(* IEC 61131-3 sources: B-R/Processes/EDT (part 3) *)

(* ---- EDTP3S2A_ACTION.st ---- *)
ACTION P3S2A_ACT:
	//设定时间
	FOR i := 0 TO EDTP3S2_STEP_NUM DO
		IF EDTP3S2A_ST[i] < T#5s THEN
			EDTP3S2A_ST[i] := T#5s;
		END_IF;
		EDTP3S2A_STEP[i].set_time := EDTP3S2A_ST[i];
	END_FOR;

	//流程步骤
	ProcessHandleFC(EDTP3S2A,EDTP3S2A_STEP[0],EDTP3S2_STEP_NUM);

	//object 手自动切换
	IF (EDTP3S2A.status.mode <> 0) AND (NOT EDTP3S2A.auto_mode_edge) THEN
		EDTP3S2A.auto_mode_edge := TRUE;
		EDTP3S2A.manual_mode_edge := FALSE;

		EDTR17A.control.auto_operate := TRUE;
		EDTXV0902.control.auto_operate := TRUE;
		EDTXV2128.control.auto_operate := TRUE;
		EDTXV2119.control.auto_operate := TRUE;
		EDTXV2121.control.auto_operate := TRUE;
		EDTTV0901C.control.auto_operate := TRUE;
		EDTTV0901D.control.auto_operate := TRUE;
		EDTTV0901E.control.auto_operate := TRUE;
		EDTTV0901F.control.auto_operate := TRUE;
		EDTTV0902B.control.auto_operate := TRUE;
		EDTTV0902A.control.auto_operate := TRUE;
		EDTTV0901A.control.auto_operate := TRUE;
		EDTTV0901B.control.auto_operate := TRUE;
		EDTXV0918.control.auto_operate := TRUE;
		EDTFQV0901.control.auto_operate := TRUE;
		EDTFQV0904.control.auto_operate := TRUE;
		EDTLV1002.control.auto_operate := TRUE;
		EDTP16.control.auto_operate := TRUE;
		EDTXV0925.control.auto_operate := TRUE;
		STFP06.control.auto_operate := TRUE;
		STFLV0601.control.auto_operate := TRUE;
		STFLV0602.control.auto_operate := TRUE;
		EDTLV1003.control.auto_operate := TRUE;
	END_IF;

	IF (EDTP3S2A.status.mode = 0) AND (NOT EDTP3S2A.manual_mode_edge) THEN
		EDTP3S2A.manual_mode_edge := TRUE;
		EDTP3S2A.auto_mode_edge := FALSE;

		EDTR17A.control.manual_operate := TRUE;
		EDTXV0902.control.manual_operate := TRUE;
		EDTXV2128.control.manual_operate := TRUE;
		EDTXV2119.control.manual_operate := TRUE;
		EDTXV2121.control.manual_operate := TRUE;
		EDTTV0901C.control.manual_operate := TRUE;
		EDTTV0901D.control.manual_operate := TRUE;
		EDTTV0901E.control.manual_operate := TRUE;
		EDTTV0901F.control.manual_operate := TRUE;
		EDTTV0902B.control.manual_operate := TRUE;
		EDTTV0902A.control.manual_operate := TRUE;
		EDTTV0901A.control.manual_operate := TRUE;
		EDTTV0901B.control.manual_operate := TRUE;
		EDTXV0918.control.manual_operate := TRUE;
		EDTFQV0901.control.manual_operate := TRUE;
		EDTFQV0904.control.manual_operate := TRUE;
		EDTLV1002.control.manual_operate := TRUE;
		EDTP16.control.manual_operate := TRUE;
		EDTXV0925.control.manual_operate := TRUE;
		STFP06.control.manual_operate := TRUE;
		STFLV0601.control.manual_operate := TRUE;
		STFLV0602.control.manual_operate := TRUE;
		EDTLV1003.control.manual_operate := TRUE;
	END_IF;

	//错误信号停机
	EDTP3S2A.input.error_signal := (EDTR17A.status.motor_status >= 2) OR (EDTXV0902.status.valve_status >= 2) OR
	(EDTXV2128.status.valve_status >= 2) OR (EDTXV2119.status.valve_status >= 2) OR (EDTP16.status.motor_status >= 2) OR
	(EDTTV0901C.status.valve_status >= 2) OR (EDTTV0901D.status.valve_status >= 2) OR (EDTXV0918.status.valve_status >= 2) OR
	(EDTTV0901E.status.valve_status >= 2) OR (EDTTV0901F.status.valve_status >= 2) OR (EDTTV0902B.status.valve_status >= 2) OR
	(EDTTV0902A.status.valve_status >= 2) OR (EDTTV0901A.status.valve_status >= 2) OR (EDTTV0901B.status.valve_status >= 2) OR
	(EDTFQV0901.status.valve_status >= 2) OR (EDTFQV0904.status.valve_status >= 2) OR (EDTLV1002.status.valve_status >= 2) OR
	(EDTXV2121.status.valve_status >= 2) OR (EDTXV0925.status.valve_status >= 2) OR (STFP06.status.motor_status >= 2) OR
	(EDTLV1003.status.valve_status >= 2) OR (STFLV0601.status.valve_status >= 2 )OR (STFLV0602.status.valve_status >= 2);

	IF EDTP3S2A.status.run_state = 1 THEN
		CASE EDTP3S2A.status.run_step OF
			0:
				IF NOT EDTP3S2A_STEP[0].done THEN
					EDTR17A.control.auto_operate := TRUE;
					EDTXV0902.control.auto_operate := TRUE;
					EDTXV2128.control.auto_operate := TRUE;
					EDTXV2119.control.auto_operate := TRUE;
					EDTXV2121.control.auto_operate := TRUE;
					EDTTV0901C.control.auto_operate := TRUE;
					EDTTV0901D.control.auto_operate := TRUE;
					EDTTV0901E.control.auto_operate := TRUE;
					EDTTV0901F.control.auto_operate := TRUE;
					EDTTV0902B.control.auto_operate := TRUE;
					EDTTV0902A.control.auto_operate := TRUE;
					EDTTV0901A.control.auto_operate := TRUE;
					EDTTV0901B.control.auto_operate := TRUE;
					EDTXV0918.control.auto_operate := TRUE;
					EDTFQV0901.control.auto_operate := TRUE;
					EDTFQV0904.control.auto_operate := TRUE;
					EDTLV1002.control.auto_operate := TRUE;
					EDTP16.control.auto_operate := TRUE;
					EDTXV0925.control.auto_operate := TRUE;
					STFP06.control.auto_operate := TRUE;
					STFLV0601.control.auto_operate := TRUE;
					STFLV0602.control.auto_operate := TRUE;
					EDTLV1003.control.auto_operate := TRUE;
					EDTP3S2A_STEP[0].done := TRUE;
				END_IF;
			1:
				EDTXV0925.input.auto_open_signal := TRUE;
				IF EDTXV0905.input.close_feedback_state THEN
					EDTR17A.input.auto_run_signal := TRUE;
					EDTXV0902.input.auto_open_signal := TRUE;
					EDTTV0902A.input.auto_open_signal := FALSE;
					EDTXV2128.input.auto_open_signal := FALSE;
					IF EDTTV0902A.input.close_feedback_state AND EDTXV2128.input.close_feedback_state THEN
						EDTTV0902B.input.auto_open_signal := TRUE;
						IF EDTR17A.input.run_feedback AND EDTXV0902.input.open_feedback_state AND EDTTV0902B.input.open_feedback_state THEN
							EDTP3S2A_STEP[1].done := TRUE;
						END_IF;
					END_IF;
				END_IF;
			2:
				CASE p3_step2_3a OF
					0:
						IF NOT EDTP3S2A_STEP[2].done THEN
							p3_step2_3a := 1;
						END_IF;
					1:
						HeatPot_1(ST1 := DINT_TO_TIME(EDTP3S2A_PARA_T1 * 1000),
						ST2 := DINT_TO_TIME(EDTP3S2A_PARA_T2 * 1000),
						V3 := EDTTV0901C,
						V4 := EDTTV0901D,
						V5 := EDTTV0901E,
						V6 := EDTTV0901F,
						done := p3_step2_3a_1_done);
						IF p3_step2_3a_1_done THEN
							p3_step2_3a_1_done := FALSE;
							p3_step2_3a := 2;
						END_IF;
					2:
						IF EDTTIT0901.status.value >= EDTP3S2A_PARA_Temp1 THEN
							p3_step2_3a := 3;
						END_IF;
					3:
						EDTTV0901C.input.auto_open_signal := FALSE;
						IF EDTTV0901C.input.close_feedback_state THEN
							p3_step2_3a := 4;
						END_IF;
					4:
						IF EDTLIT0901.status.value >= EDTP3S2A_PARA_L1 THEN
							EDTTV0902B.input.auto_open_signal := FALSE;
							EDTTV0902A.input.auto_open_signal := TRUE;
							IF EDTXV2128.input.close_feedback_state THEN
								EDTXV0918.input.auto_open_signal := TRUE;
							END_IF;
							p3_step2_3a := 5;
						END_IF;
					5:
						IF EDTXV2128.input.open_feedback_state THEN
							EDTXV0918.input.auto_open_signal := FALSE;
						END_IF;
						IF EDTTIT0901.status.value >= EDTP3S2A_PARA_Temp2 THEN
							EDTXV0918.input.auto_open_signal := FALSE;
							EDTXV2128.input.auto_open_signal := TRUE;
							EDTXV2119.input.auto_open_signal := TRUE;
							EDTXV2121.input.auto_open_signal := TRUE;
							p3_step2_3a := 0;
							EDTP3S2A_STEP[2].done := TRUE;
						END_IF;
				END_CASE;
			3:
				LiquidTransfer_12(sp_time := DINT_TO_TIME(EDTP3S2A_PARA_T4 * 1000),
				sp_accumulation := EDTP3S2A_PARA_AC1,
				done := EDTP3S2A_STEP[3].done,
				flowmeter := EDTFQIT1904);
				EDTFQV0901.input.auto_open_signal := LiquidTransfer_12.run;
			4:
				//继续回收
				IF EDTTIT0901.status.value >= EDTP3S2A_PARA_Temp3 THEN
					EDTP3S2A_STEP[4].done := TRUE;
				END_IF;
			5:
				//现场观察V83进料的是否有EDC油珠，无油珠后点击确认
			6:
				EDTTV0901D.input.auto_open_signal := FALSE;
				EDTTV0901E.input.auto_open_signal := FALSE;
				EDTTV0901F.input.auto_open_signal := TRUE;
				LiquidTransfer_16(sp_time := DINT_TO_TIME(EDTP3S2A_PARA_T5 * 1000),
				sp_accumulation := EDTP3S2A_PARA_AC2,
				done := EDTP3S2A_STEP[6].done,
				flowmeter := EDTFQIT1904);
				EDTFQV0901.input.auto_open_signal := LiquidTransfer_16.run;
			7:
				CASE p3_step2_7a OF
					0:
						IF NOT EDTP3S2A_STEP[7].done THEN
							p3_step2_7a := 1;
						END_IF;
					1:
						IF EDTTIT0901.status.value <= EDTP3S2A_PARA_Temp6 THEN
							EDTTV0901A.input.auto_open_signal := FALSE;
							EDTTV0901B.input.auto_open_signal := FALSE;
							EDTTV0901F.input.auto_open_signal := TRUE;
							p3_step2_7a := 2;
						ELSE
							EDTTV0901F.input.auto_open_signal := FALSE;
							EDTTV0901A.input.auto_open_signal := TRUE;
							EDTTV0901B.input.auto_open_signal := TRUE;
						END_IF;
					2:
						TON_60.PT := DINT_TO_TIME(EDTP3S2A_PARA_T9 * 60 * 1000);
						EDTR17A.input.auto_run_signal := FALSE;
						IF (NOT EDTR17A.input.run_feedback) THEN
							TON_60.IN := TRUE;
						END_IF;
						IF TON_60.Q THEN
							TON_60.IN := FALSE;
							p3_step2_7a := 0;
							EDTP3S2A_STEP[7].done := TRUE;
						END_IF;
				END_CASE;
				TON_60();
			8:
				//人工抽水,完毕后点击确认
			9:
				IF EDTLIT1501.status.value >= EDTP3S2A_PARA_L2 THEN
					EDTFQV0904.input.auto_open_signal := TRUE;
					EDTLV1002.input.auto_open_signal := TRUE;
					IF EDTFQV0904.input.open_feedback_state AND EDTLV1002.input.open_feedback_state THEN
						is_v52_a := TRUE;
						EDTP3S2A_STEP[9].done := TRUE;
					END_IF;
				ELSE
					STFLV0601.input.auto_open_signal := FALSE;
					STFLV0602.input.auto_open_signal := FALSE;
					EDTFQV0904.input.auto_open_signal := TRUE;
					EDTLV1003.input.auto_open_signal := TRUE;
					IF STFLV0601.input.close_feedback_state AND STFLV0602.input.close_feedback_state AND EDTFQV0904.input.open_feedback_state AND EDTLV1003.input.open_feedback_state THEN
						is_v52_a := FALSE;
						EDTP3S2A_STEP[9].done := TRUE;
					END_IF;
				END_IF;
			10:
				IF is_v52_a THEN
					LiquidTransfer_21(sp_time := DINT_TO_TIME(EDTP3S2A_PARA_T6 * 1000),
					sp_accumulation := EDTP3S2A_PARA_AC3,
					done := EDTP3S2A_STEP[10].done,
					flowmeter := EDTFQIT2101);
					EDTP16.input.auto_run_signal := LiquidTransfer_21.run;
				ELSE
					LiquidTransfer_1(sp_time := DINT_TO_TIME(EDTP3S2A_PARA_T6 * 1000),
					sp_accumulation := EDTP3S2A_PARA_AC3,
					done := EDTP3S2A_STEP[10].done,
					flowmeter := STFFQIT0602);
					STFP06.input.auto_run_signal := LiquidTransfer_1.run;
				END_IF;
			11:
				IF is_v52_a THEN
					IF EDTFQIT2101.flowrate <= flowrate_threshold THEN
						EDTFQV0904.input.auto_open_signal := FALSE;
						EDTLV1002.input.auto_open_signal := FALSE;
						EDTR17A.input.auto_run_signal := TRUE;
						IF EDTFQV0904.input.close_feedback_state AND EDTLV1002.input.close_feedback_state AND EDTR17A.input.auto_run_signal THEN
							EDTTV0901D.input.auto_open_signal := TRUE;
							EDTP3S2A_STEP[11].done := TRUE;
						END_IF;
					END_IF;
				ELSE
					IF STFFQIT0602.flowrate <= flowrate_threshold THEN
						EDTFQV0904.input.auto_open_signal := FALSE;
						EDTLV1003.input.auto_open_signal := FALSE;
						EDTR17A.input.auto_run_signal := TRUE;
						IF EDTFQV0904.input.close_feedback_state AND EDTLV1003.input.close_feedback_state AND EDTR17A.input.auto_run_signal THEN
							EDTTV0901D.input.auto_open_signal := TRUE;
							EDTP3S2A_STEP[11].done := TRUE;
						END_IF;
					END_IF;
				END_IF;

			12:
				TON_21.PT := DINT_TO_TIME(EDTP3S2A_PARA_T7 * 1000);
				IF EDTTV0901D.input.open_feedback_state THEN
					TON_21.IN := TRUE;
				END_IF;
				IF TON_21.Q THEN
					TON_21.IN := FALSE;
					EDTTV0901F.input.auto_open_signal := FALSE;
					EDTTV0901E.input.auto_open_signal := TRUE;
					EDTP3S2A_STEP[12].done := TRUE;
				END_IF;
				TON_21();
			13:
				TON_26.PT := DINT_TO_TIME(EDTP3S2A_PARA_T8 * 60 * 1000);
				IF EDTTIT0901.status.value >= EDTP3S2A_PARA_Temp4 THEN
					EDTTV0901D.input.auto_open_signal := FALSE;
					TON_26.IN := TRUE;
				END_IF;
				IF TON_26.Q THEN
					TON_26.IN := FALSE;
					EDTP3S2A_STEP[13].done := TRUE;
				END_IF;
				TON_26();
			14:
				//人工转移
			15:
				EDTR17A.input.auto_run_signal := FALSE;
				EDTTV0901E.input.auto_open_signal := FALSE;
				EDTP3S2A_STEP[15].done := TRUE;
		END_CASE;
	END_IF;

	//人工确认步骤可用
	IF (EDTP3S2A.status.run_state) AND (NOT EDTP3S2A_STEP[EDTP3S2A.status.run_step].done AND ((EDTP3S2A.status.run_step = 5)
		OR (EDTP3S2A.status.run_step = 8) OR (EDTP3S2A.status.run_step = 14))) THEN
		EDTP3S2A.status.confirm_enable := TRUE;
	ELSE
		EDTP3S2A.status.confirm_enable := FALSE;
	END_IF;
END_ACTION

(* ---- EDTP3S2B_ACTION.st ---- *)
ACTION P3S2B_ACT:
	//设定时间
	FOR i := 0 TO EDTP3S2_STEP_NUM DO
		IF EDTP3S2B_ST[i] < T#5s THEN
			EDTP3S2B_ST[i] := T#5s;
		END_IF;
		EDTP3S2B_STEP[i].set_time := EDTP3S2B_ST[i];
	END_FOR;

	//流程步骤
	ProcessHandleFC(EDTP3S2B,EDTP3S2B_STEP[0],EDTP3S2_STEP_NUM);

	//object 手自动切换
	IF (EDTP3S2B.status.mode <> 0) AND (NOT EDTP3S2B.auto_mode_edge) THEN
		EDTP3S2B.auto_mode_edge := TRUE;
		EDTP3S2B.manual_mode_edge := FALSE;

		EDTR17B.control.auto_operate := TRUE;
		EDTXV0912.control.auto_operate := TRUE;
		EDTXV2128.control.auto_operate := TRUE;
		EDTXV2119.control.auto_operate := TRUE;
		EDTXV2121.control.auto_operate := TRUE;
		EDTTV0903C.control.auto_operate := TRUE;
		EDTTV0903D.control.auto_operate := TRUE;
		EDTTV0903E.control.auto_operate := TRUE;
		EDTTV0903F.control.auto_operate := TRUE;
		EDTTV0904B.control.auto_operate := TRUE;
		EDTTV0904A.control.auto_operate := TRUE;
		EDTTV0903A.control.auto_operate := TRUE;
		EDTTV0903B.control.auto_operate := TRUE;
		EDTXV0918.control.auto_operate := TRUE;
		EDTFQV0902.control.auto_operate := TRUE;
		EDTFQV0905.control.auto_operate := TRUE;
		EDTLV1002.control.auto_operate := TRUE;
		EDTP16.control.auto_operate := TRUE;
		EDTXV0925.control.auto_operate := TRUE;
		STFP06.control.auto_operate := TRUE;
		STFLV0601.control.auto_operate := TRUE;
		STFLV0602.control.auto_operate := TRUE;
		EDTLV1003.control.auto_operate := TRUE;
	END_IF;

	IF (EDTP3S2B.status.mode = 0) AND (NOT EDTP3S2B.manual_mode_edge) THEN
		EDTP3S2B.manual_mode_edge := TRUE;
		EDTP3S2B.auto_mode_edge := FALSE;

		EDTR17B.control.manual_operate := TRUE;
		EDTXV0912.control.manual_operate := TRUE;
		EDTXV2128.control.manual_operate := TRUE;
		EDTXV2119.control.manual_operate := TRUE;
		EDTXV2121.control.manual_operate := TRUE;
		EDTTV0903C.control.manual_operate := TRUE;
		EDTTV0903D.control.manual_operate := TRUE;
		EDTTV0903E.control.manual_operate := TRUE;
		EDTTV0903F.control.manual_operate := TRUE;
		EDTTV0904B.control.manual_operate := TRUE;
		EDTTV0904A.control.manual_operate := TRUE;
		EDTTV0903A.control.manual_operate := TRUE;
		EDTTV0903B.control.manual_operate := TRUE;
		EDTXV0918.control.manual_operate := TRUE;
		EDTFQV0902.control.manual_operate := TRUE;
		EDTFQV0905.control.manual_operate := TRUE;
		EDTLV1002.control.manual_operate := TRUE;
		EDTP16.control.manual_operate := TRUE;
		EDTXV0925.control.manual_operate := TRUE;
		STFP06.control.manual_operate := TRUE;
		STFLV0601.control.manual_operate := TRUE;
		STFLV0602.control.manual_operate := TRUE;
		EDTLV1003.control.manual_operate := TRUE;
	END_IF;

	//错误信号停机
	EDTP3S2B.input.error_signal := (EDTR17B.status.motor_status >= 2) OR (EDTXV0912.status.valve_status >= 2) OR
	(EDTXV2128.status.valve_status >= 2) OR (EDTXV2119.status.valve_status >= 2) OR (EDTP16.status.motor_status >= 2) OR
	(EDTTV0903C.status.valve_status >= 2) OR (EDTTV0903D.status.valve_status >= 2) OR (EDTXV0918.status.valve_status >= 2) OR
	(EDTTV0903E.status.valve_status >= 2) OR (EDTTV0903F.status.valve_status >= 2) OR (EDTTV0904B.status.valve_status >= 2) OR
	(EDTTV0904A.status.valve_status >= 2) OR (EDTTV0903A.status.valve_status >= 2) OR (EDTTV0903B.status.valve_status >= 2) OR
	(EDTFQV0902.status.valve_status >= 2) OR (EDTFQV0905.status.valve_status >= 2) OR (EDTLV1002.status.valve_status >= 2) OR
	(EDTXV2121.status.valve_status >= 2) OR (EDTXV0925.status.valve_status >= 2) OR (STFP06.status.motor_status >= 2) OR
	(EDTLV1003.status.valve_status >= 2) OR (STFLV0601.status.valve_status >= 2 )OR (STFLV0602.status.valve_status >= 2);

	IF EDTP3S2B.status.run_state = 1 THEN
		CASE EDTP3S2B.status.run_step OF
			0:
				IF NOT EDTP3S2B_STEP[0].done THEN
					EDTR17B.control.auto_operate := TRUE;
					EDTXV0912.control.auto_operate := TRUE;
					EDTXV2128.control.auto_operate := TRUE;
					EDTXV2119.control.auto_operate := TRUE;
					EDTXV2121.control.auto_operate := TRUE;
					EDTTV0903C.control.auto_operate := TRUE;
					EDTTV0903D.control.auto_operate := TRUE;
					EDTTV0903E.control.auto_operate := TRUE;
					EDTTV0903F.control.auto_operate := TRUE;
					EDTTV0904B.control.auto_operate := TRUE;
					EDTTV0904A.control.auto_operate := TRUE;
					EDTTV0903A.control.auto_operate := TRUE;
					EDTTV0903B.control.auto_operate := TRUE;
					EDTXV0918.control.auto_operate := TRUE;
					EDTFQV0902.control.auto_operate := TRUE;
					EDTFQV0905.control.auto_operate := TRUE;
					EDTLV1002.control.auto_operate := TRUE;
					EDTP16.control.auto_operate := TRUE;
					EDTXV0925.control.auto_operate := TRUE;
					STFP06.control.auto_operate := TRUE;
					STFLV0601.control.auto_operate := TRUE;
					STFLV0602.control.auto_operate := TRUE;
					EDTLV1003.control.auto_operate := TRUE;
					EDTP3S2B_STEP[0].done := TRUE;
				END_IF;
			1:
				EDTXV0925.input.auto_open_signal := TRUE;
				IF EDTXV0913.input.close_feedback_state THEN
					EDTR17B.input.auto_run_signal := TRUE;
					EDTXV0912.input.auto_open_signal := TRUE;
					EDTTV0904A.input.auto_open_signal := FALSE;
					EDTXV2128.input.auto_open_signal := FALSE;
					IF EDTTV0904A.input.close_feedback_state AND EDTXV2128.input.close_feedback_state THEN
						EDTTV0904B.input.auto_open_signal := TRUE;
						IF EDTR17B.input.run_feedback AND EDTXV0912.input.open_feedback_state AND EDTTV0904B.input.open_feedback_state THEN
							EDTP3S2B_STEP[1].done := TRUE;
						END_IF;
					END_IF;
				END_IF;
			2:
				CASE p3_step2_3b OF
					0:
						IF NOT EDTP3S2B_STEP[2].done THEN
							p3_step2_3b := 1;
						END_IF;
					1:
						HeatPot_11(ST1 := DINT_TO_TIME(EDTP3S2B_PARA_T1 * 1000),
						ST2 := DINT_TO_TIME(EDTP3S2B_PARA_T2 * 1000),
						V3 := EDTTV0903C,
						V4 := EDTTV0903D,
						V5 := EDTTV0903E,
						V6 := EDTTV0903F,
						done := p3_step2_3b_1_done);
						IF p3_step2_3b_1_done THEN
							p3_step2_3b_1_done := FALSE;
							p3_step2_3b := 2;
						END_IF;
					2:
						IF EDTTIT0903.status.value >= EDTP3S2B_PARA_Temp1 THEN
							p3_step2_3b := 3;
						END_IF;
					3:
						EDTTV0903C.input.auto_open_signal := FALSE;
						IF EDTTV0903C.input.close_feedback_state THEN
							p3_step2_3b := 4;
						END_IF;
					4:
						IF EDTLIT0902.status.value >= EDTP3S2B_PARA_L1 THEN
							EDTTV0904B.input.auto_open_signal := FALSE;
							EDTTV0904A.input.auto_open_signal := TRUE;
							IF EDTXV2128.input.close_feedback_state THEN
								EDTXV0918.input.auto_open_signal := TRUE;
							END_IF;
							p3_step2_3b := 5;
						END_IF;
					5:
						IF EDTXV2128.input.open_feedback_state THEN
							EDTXV0918.input.auto_open_signal := FALSE;
						END_IF;
						IF EDTTIT0903.status.value >= EDTP3S2B_PARA_Temp2 THEN
							EDTXV0918.input.auto_open_signal := FALSE;
							EDTXV2128.input.auto_open_signal := TRUE;
							EDTXV2119.input.auto_open_signal := TRUE;
							EDTXV2121.input.auto_open_signal := TRUE;
							p3_step2_3b := 0;
							EDTP3S2B_STEP[2].done := TRUE;
						END_IF;
				END_CASE;
			3:
				LiquidTransfer_17(sp_time := DINT_TO_TIME(EDTP3S2B_PARA_T4 * 1000),
				sp_accumulation := EDTP3S2B_PARA_AC1,
				done := EDTP3S2B_STEP[3].done,
				flowmeter := EDTFQIT1904);
				EDTFQV0902.input.auto_open_signal := LiquidTransfer_17.run;
			4:
				//继续回收
				IF EDTTIT0903.status.value >= EDTP3S2B_PARA_Temp3 THEN
					EDTP3S2B_STEP[4].done := TRUE;
				END_IF;
			5:
				//现场观察V83进料的是否有EDC油珠，无油珠后点击确认
			6:
				EDTTV0903D.input.auto_open_signal := FALSE;
				EDTTV0903E.input.auto_open_signal := FALSE;
				EDTTV0903F.input.auto_open_signal := TRUE;
				LiquidTransfer_18(sp_time := DINT_TO_TIME(EDTP3S2B_PARA_T5 * 1000),
				sp_accumulation := EDTP3S2B_PARA_AC2,
				done := EDTP3S2B_STEP[6].done,
				flowmeter := EDTFQIT1904);
				EDTFQV0902.input.auto_open_signal := LiquidTransfer_18.run;
			7:
				CASE p3_step2_7b OF
					0:
						IF NOT EDTP3S2B_STEP[7].done THEN
							p3_step2_7b := 1;
						END_IF;
					1:
						IF EDTTIT0903.status.value <= EDTP3S2B_PARA_Temp6 THEN
							EDTTV0903A.input.auto_open_signal := FALSE;
							EDTTV0903B.input.auto_open_signal := FALSE;
							EDTTV0903F.input.auto_open_signal := TRUE;
							p3_step2_7b := 2;
						ELSE
							EDTTV0903F.input.auto_open_signal := FALSE;
							EDTTV0903A.input.auto_open_signal := TRUE;
							EDTTV0903B.input.auto_open_signal := TRUE;
						END_IF;
					2:
						TON_85.PT := DINT_TO_TIME(EDTP3S2B_PARA_T9 * 60 * 1000);
						EDTR17B.input.auto_run_signal := FALSE;
						IF (NOT EDTR17B.input.run_feedback) THEN
							TON_85.IN := TRUE;
						END_IF;
						IF TON_85.Q THEN
							TON_85.IN := FALSE;
							p3_step2_7b := 0;
							EDTP3S2B_STEP[7].done := TRUE;
						END_IF;
				END_CASE;
				TON_85();
			8:
				//人工抽水
			9:
				IF EDTLIT1501.status.value >= EDTP3S2B_PARA_L2 THEN
					EDTFQV0905.input.auto_open_signal := TRUE;
					EDTLV1002.input.auto_open_signal := TRUE;
					IF EDTFQV0905.input.open_feedback_state AND EDTLV1002.input.open_feedback_state THEN
						is_v52_b := TRUE;
						EDTP3S2B_STEP[9].done := TRUE;
					END_IF;
				ELSE
					STFLV0601.input.auto_open_signal := FALSE;
					STFLV0602.input.auto_open_signal := FALSE;
					EDTFQV0905.input.auto_open_signal := TRUE;
					EDTLV1003.input.auto_open_signal := TRUE;
					IF STFLV0601.input.close_feedback_state AND STFLV0602.input.close_feedback_state AND EDTFQV0905.input.open_feedback_state AND EDTLV1003.input.open_feedback_state THEN
						is_v52_b := FALSE;
						EDTP3S2B_STEP[9].done := TRUE;
					END_IF;
				END_IF;
			10:
				IF is_v52_b THEN
					LiquidTransfer_22(sp_time := DINT_TO_TIME(EDTP3S2B_PARA_T6 * 1000),
					sp_accumulation := EDTP3S2B_PARA_AC3,
					done := EDTP3S2B_STEP[10].done,
					flowmeter := EDTFQIT2101);
					EDTP16.input.auto_run_signal := LiquidTransfer_22.run;
				ELSE
					LiquidTransfer_2(sp_time := DINT_TO_TIME(EDTP3S2B_PARA_T6 * 1000),
					sp_accumulation := EDTP3S2B_PARA_AC3,
					done := EDTP3S2B_STEP[10].done,
					flowmeter := STFFQIT0602);
					STFP06.input.auto_run_signal := LiquidTransfer_2.run;
				END_IF;
			11:
				IF is_v52_b THEN
					IF EDTFQIT2101.flowrate <= flowrate_threshold THEN
						EDTFQV0905.input.auto_open_signal := FALSE;
						EDTLV1002.input.auto_open_signal := FALSE;
						EDTR17B.input.auto_run_signal := TRUE;
						IF EDTFQV0905.input.close_feedback_state AND EDTLV1002.input.close_feedback_state AND EDTR17B.input.auto_run_signal THEN
							EDTTV0903D.input.auto_open_signal := TRUE;
							EDTP3S2B_STEP[11].done := TRUE;
						END_IF;
					END_IF;
				ELSE
					IF STFFQIT0602.flowrate <= flowrate_threshold THEN
						EDTFQV0905.input.auto_open_signal := FALSE;
						EDTLV1003.input.auto_open_signal := FALSE;
						EDTR17B.input.auto_run_signal := TRUE;
						IF EDTFQV0905.input.close_feedback_state AND EDTLV1003.input.close_feedback_state AND EDTR17B.input.auto_run_signal THEN
							EDTTV0903D.input.auto_open_signal := TRUE;
							EDTP3S2B_STEP[11].done := TRUE;
						END_IF;
					END_IF;
				END_IF;
			12:
				TON_29.PT := DINT_TO_TIME(EDTP3S2B_PARA_T7 * 1000);
				IF EDTTV0903D.input.open_feedback_state THEN
					TON_29.IN := TRUE;
				END_IF;
				IF TON_29.Q THEN
					TON_29.IN := FALSE;
					EDTTV0903F.input.auto_open_signal := FALSE;
					EDTTV0903E.input.auto_open_signal := TRUE;
					EDTP3S2B_STEP[12].done := TRUE;
				END_IF;
				TON_29();
			13:
				TON_42.PT := DINT_TO_TIME(EDTP3S2B_PARA_T8 * 60 * 1000);
				IF EDTTIT0903.status.value >= EDTP3S2B_PARA_Temp4 THEN
					EDTTV0903D.input.auto_open_signal := FALSE;
					TON_42.IN := TRUE;
				END_IF;
				IF TON_42.Q THEN
					TON_42.IN := FALSE;
					EDTP3S2B_STEP[13].done := TRUE;
				END_IF;
				TON_42();
			14:
				//人工转移
			15:
				EDTR17B.input.auto_run_signal := FALSE;
				EDTTV0903E.input.auto_open_signal := FALSE;
				EDTP3S2B_STEP[15].done := TRUE;
		END_CASE;
	END_IF;

	//人工确认步骤可用
	IF (EDTP3S2B.status.run_state) AND (NOT EDTP3S2B_STEP[EDTP3S2B.status.run_step].done AND ((EDTP3S2B.status.run_step = 5)
		OR (EDTP3S2B.status.run_step = 8) OR (EDTP3S2B.status.run_step = 14))) THEN
		EDTP3S2B.status.confirm_enable := TRUE;
	ELSE
		EDTP3S2B.status.confirm_enable := FALSE;
	END_IF;
END_ACTION

(* ---- EDTP3S2C_ACTION.st ---- *)
ACTION P3S2C_ACT:
	//设定时间
	FOR i := 0 TO EDTP3S2_STEP_NUM DO
		IF EDTP3S2C_ST[i] < T#5s THEN
			EDTP3S2C_ST[i] := T#5s;
		END_IF;
		EDTP3S2C_STEP[i].set_time := EDTP3S2C_ST[i];
	END_FOR;

	//流程步骤
	ProcessHandleFC(EDTP3S2C,EDTP3S2C_STEP[0],EDTP3S2_STEP_NUM);

	//object 手自动切换
	IF (EDTP3S2C.status.mode <> 0) AND (NOT EDTP3S2C.auto_mode_edge) THEN
		EDTP3S2C.auto_mode_edge := TRUE;
		EDTP3S2C.manual_mode_edge := FALSE;

		EDTR20.control.auto_operate := TRUE;
		EDTXV2107.control.auto_operate := TRUE;
		EDTXV2119.control.auto_operate := TRUE;
		EDTXV2110.control.auto_operate := TRUE;
		EDTTV2101C.control.auto_operate := TRUE;
		EDTTV2101D.control.auto_operate := TRUE;
		EDTTV2101E.control.auto_operate := TRUE;
		EDTTV2101F.control.auto_operate := TRUE;
		EDTXV2111.control.auto_operate := TRUE;
		EDTXV2113.control.auto_operate := TRUE;
		EDTTV2101B.control.auto_operate := TRUE;
		EDTTV2101A.control.auto_operate := TRUE;
		EDTXV2112.control.auto_operate := TRUE;
		EDTFQV2102.control.auto_operate := TRUE;
		EDTFQV2101.control.auto_operate := TRUE;
		EDTLV1002.control.auto_operate := TRUE;
		EDTP16.control.auto_operate := TRUE;
		EDTXV2109.control.auto_operate := TRUE;
		STFP06.control.auto_operate := TRUE;
		STFLV0601.control.auto_operate := TRUE;
		STFLV0602.control.auto_operate := TRUE;
		EDTLV1003.control.auto_operate := TRUE;
	END_IF;

	IF (EDTP3S2C.status.mode = 0) AND (NOT EDTP3S2C.manual_mode_edge) THEN
		EDTP3S2C.manual_mode_edge := TRUE;
		EDTP3S2C.auto_mode_edge := FALSE;

		EDTR20.control.manual_operate := TRUE;
		EDTXV2107.control.manual_operate := TRUE;
		EDTXV2119.control.manual_operate := TRUE;
		EDTXV2110.control.manual_operate := TRUE;
		EDTTV2101C.control.manual_operate := TRUE;
		EDTTV2101D.control.manual_operate := TRUE;
		EDTTV2101E.control.manual_operate := TRUE;
		EDTTV2101F.control.manual_operate := TRUE;
		EDTXV2111.control.manual_operate := TRUE;
		EDTXV2113.control.manual_operate := TRUE;
		EDTTV2101B.control.manual_operate := TRUE;
		EDTTV2101A.control.manual_operate := TRUE;
		EDTXV2112.control.manual_operate := TRUE;
		EDTFQV2102.control.manual_operate := TRUE;
		EDTFQV2101.control.manual_operate := TRUE;
		EDTLV1002.control.manual_operate := TRUE;
		EDTXV2109.control.manual_operate := TRUE;
		EDTP16.control.manual_operate := TRUE;
		STFP06.control.manual_operate := TRUE;
		STFLV0601.control.manual_operate := TRUE;
		STFLV0602.control.manual_operate := TRUE;
		EDTLV1003.control.manual_operate := TRUE;
	END_IF;

	//错误信号停机
	EDTP3S2C.input.error_signal := (EDTR20.status.motor_status >= 2) OR (EDTXV2107.status.valve_status >= 2) OR
	(EDTXV2119.status.valve_status >= 2) OR (EDTXV2110.status.valve_status >= 2) OR (EDTP16.status.motor_status >= 2) OR
	(EDTTV2101C.status.valve_status >= 2) OR (EDTTV2101D.status.valve_status >= 2) OR (EDTXV2113.status.valve_status >= 2) OR
	(EDTTV2101E.status.valve_status >= 2) OR (EDTTV2101F.status.valve_status >= 2) OR (EDTXV2111.status.valve_status >= 2) OR
	(EDTTV2101B.status.valve_status >= 2) OR (EDTTV2101A.status.valve_status >= 2) OR (STFP06.status.motor_status >= 2) OR
	(EDTFQV2102.status.valve_status >= 2) OR (EDTFQV2101.status.valve_status >= 2) OR (EDTLV1002.status.valve_status >= 2) OR
	(EDTXV2112.status.valve_status >= 2) OR (EDTXV2109.status.valve_status >= 2 )OR (EDTLV1003.status.valve_status >= 2) OR
	(STFLV0601.status.valve_status >= 2 )OR (STFLV0602.status.valve_status >= 2);

	TON_19.PT := DINT_TO_TIME(EDTP3S2C_PARA_T3 * 60 * 1000);
	IF EDTP3S2C.status.run_state = 1 THEN
		IF EDTTIT2102.status.value >= EDTP3S2C_PARA_Temp5 THEN
			TON_19.IN := TRUE;
		END_IF;
		CASE EDTP3S2C.status.run_step OF
			0:
				IF NOT EDTP3S2C_STEP[0].done THEN
					EDTR20.control.auto_operate := TRUE;
					EDTXV2107.control.auto_operate := TRUE;
					EDTXV2119.control.auto_operate := TRUE;
					EDTXV2110.control.auto_operate := TRUE;
					EDTTV2101C.control.auto_operate := TRUE;
					EDTTV2101D.control.auto_operate := TRUE;
					EDTTV2101E.control.auto_operate := TRUE;
					EDTTV2101F.control.auto_operate := TRUE;
					EDTXV2111.control.auto_operate := TRUE;
					EDTXV2113.control.auto_operate := TRUE;
					EDTTV2101B.control.auto_operate := TRUE;
					EDTTV2101A.control.auto_operate := TRUE;
					EDTXV2112.control.auto_operate := TRUE;
					EDTFQV2102.control.auto_operate := TRUE;
					EDTFQV2101.control.auto_operate := TRUE;
					EDTLV1002.control.auto_operate := TRUE;
					EDTP16.control.auto_operate := TRUE;
					EDTXV2109.control.auto_operate := TRUE;
					STFP06.control.auto_operate := TRUE;
					STFLV0601.control.auto_operate := TRUE;
					STFLV0602.control.auto_operate := TRUE;
					EDTLV1003.control.auto_operate := TRUE;
					EDTP3S2C_STEP[0].done := TRUE;
				END_IF;
			1:
				EDTXV2109.input.auto_open_signal := TRUE;
				IF EDTXV2114.input.close_feedback_state THEN
					EDTR20.input.auto_run_signal := TRUE;
					EDTXV2107.input.auto_open_signal := TRUE;
					EDTXV2113.input.auto_open_signal := FALSE;
					IF EDTXV2113.input.close_feedback_state THEN
						EDTXV2111.input.auto_open_signal := TRUE;
						IF EDTR20.input.run_feedback AND EDTXV2107.input.open_feedback_state AND EDTXV2111.input.open_feedback_state THEN
							EDTP3S2C_STEP[1].done := TRUE;
						END_IF;
					END_IF;
				END_IF;
			2:
				CASE p3_step2_3c OF
					0:
						IF NOT EDTP3S2C_STEP[2].done THEN
							p3_step2_3c := 1;
						END_IF;
					1:
						HeatPot_15(ST1 := DINT_TO_TIME(EDTP3S2C_PARA_T1 * 1000),
						ST2 := DINT_TO_TIME(EDTP3S2C_PARA_T2 * 1000),
						V3 := EDTTV2101C,
						V4 := EDTTV2101D,
						V5 := EDTTV2101E,
						V6 := EDTTV2101F,
						done := p3_step2_3c_1_done);
						IF p3_step2_3c_1_done THEN
							p3_step2_3c_1_done := FALSE;
							p3_step2_3c := 2;
						END_IF;
					2:
						IF EDTTIT2101.status.value >= EDTP3S2C_PARA_Temp1 THEN
							p3_step2_3c := 3;
						END_IF;
					3:
						EDTTV2101C.input.auto_open_signal := FALSE;
						IF EDTTV2101C.input.close_feedback_state THEN
							p3_step2_3c := 4;
						END_IF;
					4:
						IF TON_19.Q OR EDTLSS2101.low THEN
							TON_19.IN := FALSE;
							EDTXV2111.input.auto_open_signal := FALSE;
							EDTXV2112.input.auto_open_signal := TRUE;
							p3_step2_3c := 5;
						END_IF
					5:
						IF EDTTIT2101.status.value >= EDTP3S2C_PARA_Temp2 THEN
							EDTXV2112.input.auto_open_signal := FALSE;
							EDTXV2113.input.auto_open_signal := TRUE;
							EDTXV2119.input.auto_open_signal := TRUE;
							EDTXV2110.input.auto_open_signal := TRUE;
							p3_step2_3c := 0;
							EDTP3S2C_STEP[2].done := TRUE;
						END_IF;
				END_CASE;
			3:
				LiquidTransfer_19(sp_time := DINT_TO_TIME(EDTP3S2C_PARA_T4 * 1000),
				sp_accumulation := EDTP3S2C_PARA_AC1,
				done := EDTP3S2C_STEP[3].done,
				flowmeter := EDTFQIT1904);
				EDTFQV2102.input.auto_open_signal := LiquidTransfer_19.run;
			4:
				//继续回收
				IF EDTTIT2101.status.value >= EDTP3S2C_PARA_Temp3 THEN
					EDTP3S2C_STEP[4].done := TRUE;
				END_IF;
			5:
				//现场观察V83进料的是否有EDC油珠，无油珠后点击确认
			6:
				EDTTV2101D.input.auto_open_signal := FALSE;
				EDTTV2101E.input.auto_open_signal := FALSE;
				EDTTV2101F.input.auto_open_signal := TRUE;
				LiquidTransfer_20(sp_time := DINT_TO_TIME(EDTP3S2C_PARA_T5 * 1000),
				sp_accumulation := EDTP3S2C_PARA_AC2,
				done := EDTP3S2C_STEP[6].done,
				flowmeter := EDTFQIT1904);
				EDTFQV2102.input.auto_open_signal := LiquidTransfer_20.run;
			7:
				CASE p3_step2_7c OF
					0:
						IF NOT EDTP3S2C_STEP[7].done THEN
							p3_step2_7c := 1;
						END_IF;
					1:
						IF EDTTIT2101.status.value <= EDTP3S2C_PARA_Temp6 THEN
							EDTTV2101A.input.auto_open_signal := FALSE;
							EDTTV2101B.input.auto_open_signal := FALSE;
							EDTTV2101F.input.auto_open_signal := TRUE;
							p3_step2_7c := 2;
						ELSE
							EDTTV2101F.input.auto_open_signal := FALSE;
							EDTTV2101A.input.auto_open_signal := TRUE;
							EDTTV2101B.input.auto_open_signal := TRUE;
						END_IF;
					2:
						TON_86.PT := DINT_TO_TIME(EDTP3S2C_PARA_T9 * 60 * 1000);
						EDTR20.input.auto_run_signal := FALSE;
						IF (NOT EDTR20.input.run_feedback) THEN
							TON_86.IN := TRUE;
						END_IF;
						IF TON_86.Q THEN
							TON_86.IN := FALSE;
							p3_step2_7c := 0;
							EDTP3S2C_STEP[7].done := TRUE;
						END_IF;
				END_CASE;
				TON_86();
			8:
			//人工抽水
			9:
				IF EDTLIT1501.status.value >= EDTP3S2C_PARA_L2 THEN
					EDTFQV2101.input.auto_open_signal := TRUE;
					EDTLV1002.input.auto_open_signal := TRUE;
					IF EDTFQV2101.input.open_feedback_state AND EDTLV1002.input.open_feedback_state THEN
						is_v52_c := TRUE;
						EDTP3S2C_STEP[9].done := TRUE;
					END_IF;
				ELSE
					STFLV0601.input.auto_open_signal := FALSE;
					STFLV0602.input.auto_open_signal := FALSE;
					EDTFQV2101.input.auto_open_signal := TRUE;
					EDTLV1003.input.auto_open_signal := TRUE;
					IF STFLV0601.input.close_feedback_state AND STFLV0602.input.close_feedback_state AND EDTFQV2101.input.open_feedback_state AND EDTLV1003.input.open_feedback_state THEN
						is_v52_c := FALSE;
						EDTP3S2C_STEP[9].done := TRUE;
					END_IF;
				END_IF;
			10:
				IF is_v52_c THEN
					LiquidTransfer_23(sp_time := DINT_TO_TIME(EDTP3S2C_PARA_T6 * 1000),
					sp_accumulation := EDTP3S2C_PARA_AC3,
					done := EDTP3S2C_STEP[10].done,
					flowmeter := EDTFQIT2101);
					EDTP16.input.auto_run_signal := LiquidTransfer_23.run;
				ELSE
					LiquidTransfer_7(sp_time := DINT_TO_TIME(EDTP3S2C_PARA_T6 * 1000),
					sp_accumulation := EDTP3S2C_PARA_AC3,
					done := EDTP3S2C_STEP[10].done,
					flowmeter := STFFQIT0602);
					STFP06.input.auto_run_signal := LiquidTransfer_7.run;
				END_IF;
			11:
				IF is_v52_c THEN
					IF EDTFQIT2101.flowrate <= flowrate_threshold THEN
						EDTFQV2101.input.auto_open_signal := FALSE;
						EDTLV1002.input.auto_open_signal := FALSE;
						EDTR20.input.auto_run_signal := TRUE;
						IF EDTFQV2101.input.close_feedback_state AND EDTLV1002.input.close_feedback_state AND EDTR20.input.auto_run_signal THEN
							EDTTV2101D.input.auto_open_signal := TRUE;
							EDTP3S2C_STEP[11].done := TRUE;
						END_IF;
					END_IF;
				ELSE
					IF STFFQIT0602.flowrate <= flowrate_threshold THEN
						EDTFQV2101.input.auto_open_signal := FALSE;
						EDTLV1003.input.auto_open_signal := FALSE;
						EDTR20.input.auto_run_signal := TRUE;
						IF EDTFQV2101.input.close_feedback_state AND EDTLV1003.input.close_feedback_state AND EDTR20.input.auto_run_signal THEN
							EDTTV2101D.input.auto_open_signal := TRUE;
							EDTP3S2C_STEP[11].done := TRUE;
						END_IF;
					END_IF;
				END_IF;
			12:
				TON_61.PT := DINT_TO_TIME(EDTP3S2C_PARA_T7 * 1000);
				IF EDTTV2101D.input.open_feedback_state THEN
					TON_61.IN := TRUE;
				END_IF;
				IF TON_61.Q THEN
					EDTTV2101F.input.auto_open_signal := FALSE;
					EDTTV2101E.input.auto_open_signal := TRUE;
					TON_61.IN := FALSE;
					EDTP3S2C_STEP[12].done := TRUE;
				END_IF;
				TON_61();
			13:
				TON_73.PT := DINT_TO_TIME(EDTP3S2C_PARA_T8 * 60 * 1000);
				IF EDTTIT2101.status.value >= EDTP3S2C_PARA_Temp4 THEN
					EDTTV2101D.input.auto_open_signal := FALSE;
					TON_73.IN := TRUE;
				END_IF;
				IF TON_73.Q THEN
					TON_73.IN := FALSE;
					EDTP3S2C_STEP[13].done := TRUE;
				END_IF;
				TON_73();
			14:
				//人工转移
			15:
				EDTR20.input.auto_run_signal := FALSE;
				EDTTV2101E.input.auto_open_signal := FALSE;
				EDTP3S2C_STEP[15].done := TRUE;
		END_CASE;
	END_IF;
	TON_19();

	//人工确认步骤可用
	IF (EDTP3S2C.status.run_state) AND (NOT EDTP3S2C_STEP[EDTP3S2C.status.run_step].done AND ((EDTP3S2C.status.run_step = 5)
		OR (EDTP3S2C.status.run_step = 8) OR (EDTP3S2C.status.run_step = 14))) THEN
		EDTP3S2C.status.confirm_enable := TRUE;
	ELSE
		EDTP3S2C.status.confirm_enable := FALSE;
	END_IF;
END_ACTION

(* ---- EDTP3S3A_ACTION.st ---- *)
ACTION P3S3A_ACT:
	//设定时间
	FOR i := 0 TO EDTP3S3_STEP_NUM DO
		IF EDTP3S3A_ST[i] < T#5s THEN
			EDTP3S3A_ST[i] := T#5s;
		END_IF;
		EDTP3S3A_STEP[i].set_time := EDTP3S3A_ST[i];
	END_FOR;

	//流程步骤
	ProcessHandleFC(EDTP3S3A,EDTP3S3A_STEP[0],EDTP3S3_STEP_NUM);

	//object 手自动切换
	IF (EDTP3S3A.status.mode <> 0) AND (NOT EDTP3S3A.auto_mode_edge) THEN
		EDTP3S3A.auto_mode_edge := TRUE;
		EDTP3S3A.manual_mode_edge := FALSE;

		EDTXV0925.control.auto_operate := TRUE;
		EDTXV2121.control.auto_operate := TRUE;
		EDTXV2119.control.auto_operate := TRUE;
		EDTXV2126.control.auto_operate := TRUE;
		EDTP34.control.auto_operate := TRUE;
		EDTTV0901C.control.auto_operate := TRUE;
		EDTTV0901D.control.auto_operate := TRUE;
		EDTTV0901E.control.auto_operate := TRUE;
		EDTTV0901F.control.auto_operate := TRUE;
		EDTTV0901A.control.auto_operate := TRUE;
		EDTTV0901B.control.auto_operate := TRUE;
		EDTXV0923.control.auto_operate := TRUE;
		EDTXV2118.control.auto_operate := TRUE;
		EDTXV2128.control.auto_operate := TRUE;
		EDTTV0902A.control.auto_operate := TRUE;
		EDTXV0902.control.auto_operate := TRUE;
		EDTR17A.control.auto_operate := TRUE;
		EDTXV2127.control.auto_operate := TRUE;
	END_IF;

	IF (EDTP3S3A.status.mode = 0) AND (NOT EDTP3S3A.manual_mode_edge) THEN
		EDTP3S3A.manual_mode_edge := TRUE;
		EDTP3S3A.auto_mode_edge := FALSE;

		EDTXV0925.control.manual_operate := TRUE;
		EDTXV2121.control.manual_operate := TRUE;
		EDTXV2119.control.manual_operate := TRUE;
		EDTXV2126.control.manual_operate := TRUE;
		EDTP34.control.manual_operate := TRUE;
		EDTTV0901C.control.manual_operate := TRUE;
		EDTTV0901D.control.manual_operate := TRUE;
		EDTTV0901E.control.manual_operate := TRUE;
		EDTTV0901F.control.manual_operate := TRUE;
		EDTTV0901A.control.manual_operate := TRUE;
		EDTTV0901B.control.manual_operate := TRUE;
		EDTXV0923.control.manual_operate := TRUE;
		EDTXV2118.control.manual_operate := TRUE;
		EDTXV2128.control.manual_operate := TRUE;
		EDTTV0902A.control.manual_operate := TRUE;
		EDTXV0902.control.manual_operate := TRUE;
		EDTR17A.control.manual_operate := TRUE;
		EDTXV2127.control.manual_operate := TRUE;
	END_IF;

	//错误信号停机
	EDTP3S3A.input.error_signal := (EDTP34.status.motor_status >= 2) OR (EDTXV0925.status.valve_status >= 2) OR
	(EDTXV2121.status.valve_status >= 2) OR (EDTXV2119.status.valve_status >= 2) OR (EDTXV2126.status.valve_status >= 2) OR
	(EDTTV0901C.status.valve_status >= 2) OR (EDTTV0901D.status.valve_status >= 2) OR (EDTXV2128.status.valve_status >= 2) OR (EDTTV0902A.status.valve_status >= 2) OR
	(EDTTV0901E.status.valve_status >= 2) OR (EDTTV0901F.status.valve_status >= 2) OR (EDTTV0901A.status.valve_status >= 2) OR (EDTXV2127.status.valve_status >= 2) OR
	(EDTTV0901B.status.valve_status >= 2) OR (EDTXV0923.status.valve_status >= 2) OR (EDTXV2118.status.valve_status >= 2) OR (EDTXV0902.status.valve_status >= 2) OR
	(EDTR17A.status.motor_status >= 2);

	IF EDTP3S3A.status.run_state = 1 THEN
		CASE EDTP3S3A.status.run_step OF
			0:
				IF NOT EDTP3S3A_STEP[0].done THEN
					EDTXV0925.control.auto_operate := TRUE;
					EDTXV2121.control.auto_operate := TRUE;
					EDTXV2119.control.auto_operate := TRUE;
					EDTXV2126.control.auto_operate := TRUE;
					EDTP34.control.auto_operate := TRUE;
					EDTTV0901C.control.auto_operate := TRUE;
					EDTTV0901D.control.auto_operate := TRUE;
					EDTTV0901E.control.auto_operate := TRUE;
					EDTTV0901F.control.auto_operate := TRUE;
					EDTTV0901A.control.auto_operate := TRUE;
					EDTTV0901B.control.auto_operate := TRUE;
					EDTXV0923.control.auto_operate := TRUE;
					EDTXV2118.control.auto_operate := TRUE;
					EDTXV2128.control.auto_operate := TRUE;
					EDTTV0902A.control.auto_operate := TRUE;
					EDTXV0902.control.auto_operate := TRUE;
					EDTR17A.control.auto_operate := TRUE;
					EDTXV2127.control.auto_operate := TRUE;
					EDTP3S3A_STEP[0].done := TRUE;
				END_IF;
			1:
				EDTXV0925.input.auto_open_signal := FALSE;
				EDTXV2121.input.auto_open_signal := TRUE;
				EDTXV2119.input.auto_open_signal := TRUE;
				EDTXV2126.input.auto_open_signal := TRUE;
				EDTR17A.input.auto_run_signal := TRUE;
				IF EDTR17A.input.run_feedback AND EDTXV0925.input.close_feedback_state AND EDTXV2121.input.open_feedback_state AND EDTXV2119.input.open_feedback_state AND EDTXV2126.input.open_feedback_state THEN
					EDTP3S3A_STEP[1].done := TRUE;
				END_IF;
			2:
				//现场确认P34循环水手阀开启
				EDTXV2127.input.auto_open_signal := TRUE;
			3:
				EDTP34.input.auto_run_signal := TRUE;
				IF EDTP34.input.run_feedback THEN
					EDTP3S3A_STEP[3].done := TRUE;
				END_IF;
			4:
				CASE p3_step3_4a OF
					0:
						IF NOT EDTP3S3A_STEP[4].done THEN
							p3_step3_4a := 1;
						END_IF;
					1:
						IF EDTPIT0903.status.value <= EDTP3S3_PARA_P2 THEN
							p3_step3_4a := 2;
						END_IF;
					2:
						HeatPot_16(ST1 := DINT_TO_TIME(EDTP3S3_PARA_T1 * 1000),
						ST2 := DINT_TO_TIME(EDTP3S3_PARA_T2 * 1000),
						V3 := EDTTV0901C,
						V4 := EDTTV0901D,
						V5 := EDTTV0901E,
						V6 := EDTTV0901F,
						done := p3_step3_4a_1_done);
						IF p3_step3_4a_1_done THEN
							p3_step3_4a_1_done := FALSE;
							p3_step3_4a := 3;
						END_IF;
					3:
						IF EDTTIT0901.status.value >= EDTP3S3_PARA_Temp1 THEN
							p3_step3_4a := 4;
						END_IF;
					4:
						EDTTV0901C.input.auto_open_signal := FALSE;
						IF EDTTV0901C.input.close_feedback_state THEN
							p3_step3_4a := 5;
						END_IF;
					5:
						TON_20.PT := DINT_TO_TIME(EDTP3S3_PARA_T3 * 60 * 1000);
						TON_20.IN := TRUE;
						IF TON_20.Q THEN
							TON_20.IN := FALSE;
							p3_step3_4a := 6;
						END_IF;
					6:
						IF (NOT EDTP3S3B.status.run_state) AND (NOT EDTP3S3C.status.run_state) THEN
							p3_step3_4a := 7;
						ELSIF EDTP3S3B.status.run_state AND (NOT EDTP3S3C.status.run_state) THEN
							IF p3_step3_4b >= 6 THEN
								p3_step3_4a := 7;
							END_IF;
						ELSIF (NOT EDTP3S3B.status.run_state) AND  EDTP3S3C.status.run_state THEN
							IF p3_step3_4c >= 6 THEN
								p3_step3_4a := 7;
							END_IF;
						ELSIF EDTP3S3B.status.run_state AND EDTP3S3C.status.run_state THEN
							IF (p3_step3_4b >= 6) AND (p3_step3_4c >= 6) THEN
								p3_step3_4a := 7;
							END_IF;
						END_IF;
					7:
						CoolPot_9(
							time := cool_pot_time,
							V1 := EDTTV0901A,
							V2 := EDTTV0901B,
							V3 := EDTTV0901F,
							V4 := EDTTV0901D,
							V5 := EDTTV0901E,
							done := p3_step3_4a_5_done);
						IF p3_step3_4a_5_done THEN
							p3_step3_4a_5_done := FALSE;
							p3_step3_4a := 8;
						END_IF;
					8:
						IF EDTTIT0901.status.value <= EDTP3S3_PARA_Temp2 THEN
							EDTXV2121.input.auto_open_signal := FALSE;
							IF EDTXV2121.input.close_feedback_state THEN
								EDTXV0923.input.auto_open_signal := TRUE;
								EDTXV2118.input.auto_open_signal := TRUE;
								IF EDTXV0923.input.open_feedback_state AND EDTXV2118.input.open_feedback_state THEN
									p3_step3_4a := 9;
								END_IF;
							END_IF;
						END_IF;
					9:
						IF EDTPIT0903.status.value >= EDTP3S3_PARA_P1 THEN
							p3_step3_4a := 10;
						END_IF;
					10:
						EDTXV2118.input.auto_open_signal := FALSE;
						EDTXV0923.input.auto_open_signal := FALSE;
						EDTXV0925.input.auto_open_signal := TRUE;
						EDTTV0901A.input.auto_open_signal := FALSE;
						EDTTV0901B.input.auto_open_signal := FALSE;
						IF EDTXV2118.input.close_feedback_state AND EDTXV0923.input.close_feedback_state AND EDTXV0925.input.open_feedback_state AND EDTTV0901A.input.close_feedback_state AND EDTTV0901B.input.close_feedback_state THEN
							p3_step3_4a := 11;
						END_IF;
					11:
						EDTP34.input.auto_run_signal := FALSE;
						EDTXV0902.input.auto_open_signal := FALSE;
						EDTXV2119.input.auto_open_signal := FALSE;
						EDTXV2126.input.auto_open_signal := FALSE;
						EDTXV2128.input.auto_open_signal := FALSE;
						EDTR17A.input.auto_run_signal := FALSE;
						EDTTV0902A.input.auto_open_signal := FALSE;
						IF EDTXV0902.input.close_feedback_state AND EDTXV2128.input.close_feedback_state AND EDTTV0902A.input.close_feedback_state AND EDTXV2119.input.close_feedback_state
							AND EDTXV2126.input.close_feedback_state AND (NOT EDTP34.input.run_feedback) AND (NOT EDTR17A.input.run_feedback) THEN
							EDTP3S3A_STEP[4].done := TRUE;
							p3_step3_4a := 0;
						END_IF;
				END_CASE;
				TON_20();
			5:
			//现场关闭P34循环水手阀
			EDTXV2127.input.auto_open_signal := FALSE;
		END_CASE;
	END_IF;

	//人工确认步骤可用
	IF (EDTP3S3A.status.run_state) AND (NOT EDTP3S3A_STEP[EDTP3S3A.status.run_step].done AND ((EDTP3S3A.status.run_step = 2) OR (EDTP3S3A.status.run_step = 5))) THEN
		EDTP3S3A.status.confirm_enable := TRUE;
	ELSE
		EDTP3S3A.status.confirm_enable := FALSE;
	END_IF;
END_ACTION

(* ---- EDTP3S3B_ACTION.st ---- *)
ACTION P3S3B_ACT:
	//设定时间
	FOR i := 0 TO EDTP3S3_STEP_NUM DO
		IF EDTP3S3B_ST[i] < T#5s THEN
			EDTP3S3B_ST[i] := T#5s;
		END_IF;
		EDTP3S3B_STEP[i].set_time := EDTP3S3B_ST[i];
	END_FOR;

	//流程步骤
	ProcessHandleFC(EDTP3S3B,EDTP3S3B_STEP[0],EDTP3S3_STEP_NUM);

	//object 手自动切换
	IF (EDTP3S3B.status.mode <> 0) AND (NOT EDTP3S3B.auto_mode_edge) THEN
		EDTP3S3B.auto_mode_edge := TRUE;
		EDTP3S3B.manual_mode_edge := FALSE;

		EDTXV0925.control.auto_operate := TRUE;
		EDTXV2121.control.auto_operate := TRUE;
		EDTXV2119.control.auto_operate := TRUE;
		EDTXV2126.control.auto_operate := TRUE;
		EDTP34.control.auto_operate := TRUE;
		EDTTV0903C.control.auto_operate := TRUE;
		EDTTV0903D.control.auto_operate := TRUE;
		EDTTV0903E.control.auto_operate := TRUE;
		EDTTV0903F.control.auto_operate := TRUE;
		EDTTV0903A.control.auto_operate := TRUE;
		EDTTV0903B.control.auto_operate := TRUE;
		EDTXV0924.control.auto_operate := TRUE;
		EDTXV2118.control.auto_operate := TRUE;
		EDTXV2128.control.auto_operate := TRUE;
		EDTTV0904A.control.auto_operate := TRUE;
		EDTXV0912.control.auto_operate := TRUE;
		EDTR17B.control.auto_operate := TRUE;
		EDTXV2127.control.auto_operate := TRUE;
	END_IF;

	IF (EDTP3S3B.status.mode = 0) AND (NOT EDTP3S3B.manual_mode_edge) THEN
		EDTP3S3B.manual_mode_edge := TRUE;
		EDTP3S3B.auto_mode_edge := FALSE;

		EDTXV0925.control.manual_operate := TRUE;
		EDTXV2121.control.manual_operate := TRUE;
		EDTXV2119.control.manual_operate := TRUE;
		EDTXV2126.control.manual_operate := TRUE;
		EDTP34.control.manual_operate := TRUE;
		EDTTV0903C.control.manual_operate := TRUE;
		EDTTV0903D.control.manual_operate := TRUE;
		EDTTV0903E.control.manual_operate := TRUE;
		EDTTV0903F.control.manual_operate := TRUE;
		EDTTV0903A.control.manual_operate := TRUE;
		EDTTV0903B.control.manual_operate := TRUE;
		EDTXV0924.control.manual_operate := TRUE;
		EDTXV2118.control.manual_operate := TRUE;
		EDTXV2128.control.manual_operate := TRUE;
		EDTTV0904A.control.manual_operate := TRUE;
		EDTXV0912.control.manual_operate := TRUE;
		EDTR17B.control.manual_operate := TRUE;
		EDTXV2127.control.manual_operate := TRUE;
	END_IF;

	//错误信号停机
	EDTP3S3B.input.error_signal := (EDTP34.status.motor_status >= 2) OR (EDTXV0925.status.valve_status >= 2) OR
	(EDTXV2121.status.valve_status >= 2) OR (EDTXV2119.status.valve_status >= 2) OR (EDTXV2126.status.valve_status >= 2) OR
	(EDTTV0903C.status.valve_status >= 2) OR (EDTTV0903D.status.valve_status >= 2) OR (EDTXV2128.status.valve_status >= 2) OR (EDTTV0904A.status.valve_status >= 2) OR
	(EDTTV0903E.status.valve_status >= 2) OR (EDTTV0903F.status.valve_status >= 2) OR (EDTTV0903A.status.valve_status >= 2) OR (EDTXV2127.status.valve_status >= 2) OR
	(EDTTV0903B.status.valve_status >= 2) OR (EDTXV0924.status.valve_status >= 2) OR (EDTXV2118.status.valve_status >= 2) OR (EDTXV0912.status.valve_status >= 2) OR
	(EDTR17B.status.motor_status >= 2);

	IF EDTP3S3B.status.run_state = 1 THEN
		CASE EDTP3S3B.status.run_step OF
			0:
				IF NOT EDTP3S3B_STEP[0].done THEN
					EDTXV0925.control.auto_operate := TRUE;
					EDTXV2121.control.auto_operate := TRUE;
					EDTXV2119.control.auto_operate := TRUE;
					EDTXV2126.control.auto_operate := TRUE;
					EDTP34.control.auto_operate := TRUE;
					EDTTV0903C.control.auto_operate := TRUE;
					EDTTV0903D.control.auto_operate := TRUE;
					EDTTV0903E.control.auto_operate := TRUE;
					EDTTV0903F.control.auto_operate := TRUE;
					EDTTV0903A.control.auto_operate := TRUE;
					EDTTV0903B.control.auto_operate := TRUE;
					EDTXV0924.control.auto_operate := TRUE;
					EDTXV2118.control.auto_operate := TRUE;
					EDTXV2128.control.auto_operate := TRUE;
					EDTTV0904A.control.auto_operate := TRUE;
					EDTXV0912.control.auto_operate := TRUE;
					EDTR17B.control.auto_operate := TRUE;
					EDTXV2127.control.auto_operate := TRUE;
					EDTP3S3B_STEP[0].done := TRUE;
				END_IF;
			1:
				EDTR17B.input.auto_run_signal := TRUE;
				EDTXV0925.input.auto_open_signal := FALSE;
				EDTXV2121.input.auto_open_signal := TRUE;
				EDTXV2119.input.auto_open_signal := TRUE;
				EDTXV2126.input.auto_open_signal := TRUE;
				IF EDTR17B.input.run_feedback AND EDTXV0925.input.close_feedback_state AND EDTXV2121.input.open_feedback_state AND EDTXV2119.input.open_feedback_state AND EDTXV2126.input.open_feedback_state THEN
					EDTP3S3B_STEP[1].done := TRUE;
				END_IF;
			2:
				//现场确认P34循环水手阀开启
				EDTXV2127.input.auto_open_signal := TRUE;
			3:
				EDTP34.input.auto_run_signal := TRUE;
				IF EDTP34.input.run_feedback THEN
					EDTP3S3B_STEP[3].done := TRUE;
				END_IF;
			4:
				CASE p3_step3_4b OF
					0:
						IF NOT EDTP3S3B_STEP[4].done THEN
							p3_step3_4b := 1;
						END_IF;
					1:
						IF EDTPIT0904.status.value <= EDTP3S3_PARA_P2 THEN
							p3_step3_4b := 2;
						END_IF;
					2:
						HeatPot_17(ST1 := DINT_TO_TIME(EDTP3S3_PARA_T1 * 1000),
						ST2 := DINT_TO_TIME(EDTP3S3_PARA_T2 * 1000),
						V3 := EDTTV0903C,
						V4 := EDTTV0903D,
						V5 := EDTTV0903E,
						V6 := EDTTV0903F,
						done := p3_step3_4b_1_done);
						IF p3_step3_4b_1_done THEN
							p3_step3_4b_1_done := FALSE;
							p3_step3_4b := 3;
						END_IF;
					3:
						IF EDTTIT0903.status.value >= EDTP3S3_PARA_Temp1 THEN
							p3_step3_4b := 4;
						END_IF;
					4:
						EDTTV0903C.input.auto_open_signal := FALSE;
						IF EDTTV0903C.input.close_feedback_state THEN
							p3_step3_4b := 5;
						END_IF;
					5:
						TON_22.PT := DINT_TO_TIME(EDTP3S3_PARA_T3 * 60 * 1000);
						TON_22.IN := TRUE;
						IF TON_22.Q THEN
							TON_22.IN := FALSE;
							p3_step3_4b := 6;
						END_IF;
					6:
						IF (NOT EDTP3S3A.status.run_state) AND (NOT EDTP3S3C.status.run_state) THEN
							p3_step3_4b := 7;
						ELSIF EDTP3S3A.status.run_state AND (NOT EDTP3S3C.status.run_state) THEN
							IF p3_step3_4a >= 6 THEN
								p3_step3_4b := 7;
							END_IF;
						ELSIF (NOT EDTP3S3A.status.run_state) AND  EDTP3S3C.status.run_state THEN
							IF p3_step3_4c >= 6 THEN
								p3_step3_4b := 7;
							END_IF;
						ELSIF EDTP3S3A.status.run_state AND EDTP3S3C.status.run_state THEN
							IF (p3_step3_4a >= 6) AND (p3_step3_4c >= 6) THEN
								p3_step3_4b := 7;
							END_IF;
						END_IF;
					7:
						CoolPot_10(
							time := cool_pot_time,
							V1 := EDTTV0903A,
							V2 := EDTTV0903B,
							V3 := EDTTV0903F,
							V4 := EDTTV0903D,
							V5 := EDTTV0903E,
							done := p3_step3_4b_5_done);
						IF p3_step3_4b_5_done THEN
							p3_step3_4b_5_done := FALSE;
							p3_step3_4b := 8;
						END_IF;
					8:
						IF EDTTIT0903.status.value <= EDTP3S3_PARA_Temp2 THEN
							EDTXV2121.input.auto_open_signal := FALSE;
							IF EDTXV2121.input.close_feedback_state THEN
								EDTXV0924.input.auto_open_signal := TRUE;
								EDTXV2118.input.auto_open_signal := TRUE;
								IF EDTXV0924.input.open_feedback_state AND EDTXV2118.input.open_feedback_state THEN
									p3_step3_4b := 9;
								END_IF;
							END_IF;
						END_IF;
					9:
						IF EDTPIT0904.status.value >= EDTP3S3_PARA_P1 THEN
							p3_step3_4b := 10;
						END_IF;
					10:
						EDTXV2118.input.auto_open_signal := FALSE;
						EDTXV0924.input.auto_open_signal := FALSE;
						EDTXV0925.input.auto_open_signal := TRUE;
						EDTTV0903A.input.auto_open_signal := FALSE;
						EDTTV0903B.input.auto_open_signal := FALSE;
						IF EDTXV2118.input.close_feedback_state AND EDTXV0924.input.close_feedback_state AND EDTXV0925.input.open_feedback_state AND EDTTV0903A.input.close_feedback_state AND EDTTV0903B.input.close_feedback_state THEN
							p3_step3_4b := 11;
						END_IF;
					11:
						EDTP34.input.auto_run_signal := FALSE;
						EDTXV2119.input.auto_open_signal := FALSE;
						EDTXV2126.input.auto_open_signal := FALSE;
						EDTXV2128.input.auto_open_signal := FALSE;
						EDTTV0904A.input.auto_open_signal := FALSE;
						EDTXV0912.input.auto_open_signal := FALSE;
						EDTR17B.input.auto_run_signal := FALSE;
						IF EDTXV0912.input.close_feedback_state AND EDTXV2128.input.close_feedback_state AND EDTTV0904A.input.close_feedback_state
							AND EDTXV2119.input.close_feedback_state AND EDTXV2126.input.close_feedback_state AND (NOT EDTP34.input.run_feedback) AND (NOT EDTR17B.input.run_feedback) THEN
							EDTP3S3B_STEP[4].done := TRUE;
							p3_step3_4b := 0;
						END_IF;
				END_CASE;
				TON_22();
			5:
			//现场关闭P34循环水手阀
			EDTXV2127.input.auto_open_signal := FALSE;
		END_CASE;
	END_IF;

	//人工确认步骤可用
	IF (EDTP3S3B.status.run_state) AND (NOT EDTP3S3B_STEP[EDTP3S3B.status.run_step].done AND ((EDTP3S3B.status.run_step = 2) OR (EDTP3S3B.status.run_step = 5))) THEN
		EDTP3S3B.status.confirm_enable := TRUE;
	ELSE
		EDTP3S3B.status.confirm_enable := FALSE;
	END_IF;
END_ACTION

(* ---- EDTP3S3C_ACTION.st ---- *)
ACTION P3S3C_ACT:
	//设定时间
	FOR i := 0 TO EDTP3S3_STEP_NUM DO
		IF EDTP3S3C_ST[i] < T#5s THEN
			EDTP3S3C_ST[i] := T#5s;
		END_IF;
		EDTP3S3C_STEP[i].set_time := EDTP3S3C_ST[i];
	END_FOR;

	//流程步骤
	ProcessHandleFC(EDTP3S3C,EDTP3S3C_STEP[0],EDTP3S3_STEP_NUM);

	//object 手自动切换
	IF (EDTP3S3C.status.mode <> 0) AND (NOT EDTP3S3C.auto_mode_edge) THEN
		EDTP3S3C.auto_mode_edge := TRUE;
		EDTP3S3C.manual_mode_edge := FALSE;

		EDTXV2109.control.auto_operate := TRUE;
		EDTXV2110.control.auto_operate := TRUE;
		EDTXV2119.control.auto_operate := TRUE;
		EDTXV2126.control.auto_operate := TRUE;
		EDTP34.control.auto_operate := TRUE;
		EDTTV2101C.control.auto_operate := TRUE;
		EDTTV2101D.control.auto_operate := TRUE;
		EDTTV2101E.control.auto_operate := TRUE;
		EDTTV2101F.control.auto_operate := TRUE;
		EDTTV2101B.control.auto_operate := TRUE;
		EDTTV2101A.control.auto_operate := TRUE;
		EDTXV2106.control.auto_operate := TRUE;
		EDTXV2118.control.auto_operate := TRUE;
		EDTXV2113.control.auto_operate := TRUE;
		EDTXV2107.control.auto_operate := TRUE;
		EDTR20.control.auto_operate := TRUE;
		EDTXV2127.control.auto_operate := TRUE;
	END_IF;

	IF (EDTP3S3C.status.mode = 0) AND (NOT EDTP3S3C.manual_mode_edge) THEN
		EDTP3S3C.manual_mode_edge := TRUE;
		EDTP3S3C.auto_mode_edge := FALSE;

		EDTXV2109.control.manual_operate := TRUE;
		EDTXV2110.control.manual_operate := TRUE;
		EDTXV2119.control.manual_operate := TRUE;
		EDTXV2126.control.manual_operate := TRUE;
		EDTP34.control.manual_operate := TRUE;
		EDTTV2101C.control.manual_operate := TRUE;
		EDTTV2101D.control.manual_operate := TRUE;
		EDTTV2101E.control.manual_operate := TRUE;
		EDTTV2101F.control.manual_operate := TRUE;
		EDTTV2101B.control.manual_operate := TRUE;
		EDTTV2101A.control.manual_operate := TRUE;
		EDTXV2106.control.manual_operate := TRUE;
		EDTXV2118.control.manual_operate := TRUE;
		EDTXV2113.control.manual_operate := TRUE;
		EDTXV2107.control.manual_operate := TRUE;
		EDTR20.control.manual_operate := TRUE;
		EDTXV2127.control.manual_operate := TRUE;
	END_IF;

	//错误信号停机
	EDTP3S3C.input.error_signal := (EDTP34.status.motor_status >= 2) OR (EDTXV2109.status.valve_status >= 2) OR
	(EDTXV2110.status.valve_status >= 2) OR (EDTXV2119.status.valve_status >= 2) OR (EDTXV2126.status.valve_status >= 2) OR
	(EDTTV2101C.status.valve_status >= 2) OR (EDTTV2101D.status.valve_status >= 2) OR (EDTXV2113.status.valve_status >= 2) OR
	(EDTTV2101E.status.valve_status >= 2) OR (EDTTV2101F.status.valve_status >= 2) OR (EDTTV2101B.status.valve_status >= 2) OR (EDTXV2127.status.valve_status >= 2) OR
	(EDTTV2101A.status.valve_status >= 2) OR (EDTXV2106.status.valve_status >= 2) OR (EDTXV2118.status.valve_status >= 2) OR (EDTXV2107.status.valve_status >= 2) OR
	(EDTR20.status.motor_status >= 2);

	IF EDTP3S3C.status.run_state = 1 THEN
		CASE EDTP3S3C.status.run_step OF
			0:
				IF NOT EDTP3S3C_STEP[0].done THEN
					EDTXV2109.control.auto_operate := TRUE;
					EDTXV2110.control.auto_operate := TRUE;
					EDTXV2119.control.auto_operate := TRUE;
					EDTXV2126.control.auto_operate := TRUE;
					EDTP34.control.auto_operate := TRUE;
					EDTTV2101C.control.auto_operate := TRUE;
					EDTTV2101D.control.auto_operate := TRUE;
					EDTTV2101E.control.auto_operate := TRUE;
					EDTTV2101F.control.auto_operate := TRUE;
					EDTTV2101B.control.auto_operate := TRUE;
					EDTTV2101A.control.auto_operate := TRUE;
					EDTXV2106.control.auto_operate := TRUE;
					EDTXV2118.control.auto_operate := TRUE;
					EDTXV2113.control.auto_operate := TRUE;
					EDTXV2107.control.auto_operate := TRUE;
					EDTR20.control.auto_operate := TRUE;
					EDTXV2127.control.auto_operate := TRUE;
					EDTP3S3C_STEP[0].done := TRUE;
				END_IF;
			1:
				EDTXV2109.input.auto_open_signal := FALSE;
				EDTXV2110.input.auto_open_signal := TRUE;
				EDTXV2119.input.auto_open_signal := TRUE;
				EDTXV2126.input.auto_open_signal := TRUE;
				EDTR20.input.auto_run_signal := TRUE;
				IF EDTR20.input.run_feedback AND EDTXV2109.input.close_feedback_state AND EDTXV2110.input.open_feedback_state AND EDTXV2119.input.open_feedback_state AND EDTXV2126.input.open_feedback_state THEN
					EDTP3S3C_STEP[1].done := TRUE;
				END_IF;
			2:
				//现场确认P34循环水手阀开启
				EDTXV2127.input.auto_open_signal := TRUE;
			3:
				EDTP34.input.auto_run_signal := TRUE;
				IF EDTP34.input.run_feedback THEN
					EDTP3S3C_STEP[3].done := TRUE;
				END_IF;
			4:
				CASE p3_step3_4c OF
					0:
						IF NOT EDTP3S3C_STEP[4].done THEN
							p3_step3_4c := 1;
						END_IF;
					1:
						IF EDTPIT2101.status.value <= EDTP3S3_PARA_P2 THEN
							p3_step3_4c := 2;
						END_IF;
					2:
						HeatPot_18(ST1 := DINT_TO_TIME(EDTP3S3_PARA_T1 * 1000),
						ST2 := DINT_TO_TIME(EDTP3S3_PARA_T2 * 1000),
						V3 := EDTTV2101C,
						V4 := EDTTV2101D,
						V5 := EDTTV2101E,
						V6 := EDTTV2101F,
						done := p3_step3_4c_1_done);
						IF p3_step3_4c_1_done THEN
							p3_step3_4c_1_done := FALSE;
							p3_step3_4c := 3;
						END_IF;
					3:
						IF EDTTIT2101.status.value >= EDTP3S3_PARA_Temp1 THEN
							p3_step3_4c := 4;
						END_IF;
					4:
						EDTTV2101C.input.auto_open_signal := FALSE;
						IF EDTTV2101C.input.close_feedback_state THEN
							p3_step3_4c := 5;
						END_IF;
					5:
						TON_23.PT := DINT_TO_TIME(EDTP3S3_PARA_T3 * 60 * 1000);
						TON_23.IN := TRUE;
						IF TON_23.Q THEN
							TON_23.IN := FALSE;
							p3_step3_4c := 6;
						END_IF;
					6:
						IF (NOT EDTP3S3A.status.run_state) AND (NOT EDTP3S3B.status.run_state) THEN
							p3_step3_4c := 7;
						ELSIF EDTP3S3A.status.run_state AND (NOT EDTP3S3B.status.run_state) THEN
							IF p3_step3_4a >= 6 THEN
								p3_step3_4c := 7;
							END_IF;
						ELSIF (NOT EDTP3S3A.status.run_state) AND  EDTP3S3B.status.run_state THEN
							IF p3_step3_4b >= 6 THEN
								p3_step3_4c := 7;
							END_IF;
						ELSIF EDTP3S3A.status.run_state AND EDTP3S3B.status.run_state THEN
							IF (p3_step3_4a >= 6) AND (p3_step3_4b >= 6) THEN
								p3_step3_4c := 7;
							END_IF;
						END_IF;
					7:
						CoolPot_11(
							time := cool_pot_time,
							V1 := EDTTV2101B,
							V2 := EDTTV2101A,
							V3 := EDTTV2101F,
							V4 := EDTTV2101D,
							V5 := EDTTV2101E,
							done := p3_step3_4c_5_done);
						IF p3_step3_4c_5_done THEN
							p3_step3_4c_5_done := FALSE;
							p3_step3_4c := 8;
						END_IF;
					8:
						IF EDTTIT2101.status.value <= EDTP3S3_PARA_Temp2 THEN
							EDTXV2110.input.auto_open_signal := FALSE;
							IF EDTXV2110.input.close_feedback_state THEN
								EDTXV2106.input.auto_open_signal := TRUE;
								EDTXV2118.input.auto_open_signal := TRUE;
								IF EDTXV2106.input.open_feedback_state AND EDTXV2118.input.open_feedback_state THEN
									p3_step3_4c := 9;
								END_IF;
							END_IF;
						END_IF;
					9:
						IF EDTPIT2101.status.value >= EDTP3S3_PARA_P1 THEN
							p3_step3_4c := 10;
						END_IF;
					10:
						EDTXV2106.input.auto_open_signal := FALSE;
						EDTXV2118.input.auto_open_signal := FALSE;
						EDTXV2109.input.auto_open_signal := TRUE;
						EDTTV2101B.input.auto_open_signal := FALSE;
						EDTTV2101A.input.auto_open_signal := FALSE;
						IF EDTXV2118.input.close_feedback_state AND EDTXV2106.input.close_feedback_state AND EDTXV2109.input.open_feedback_state AND EDTTV2101B.input.close_feedback_state AND EDTTV2101A.input.close_feedback_state THEN
							p3_step3_4c := 11;
						END_IF;
					11:
						EDTP34.input.auto_run_signal := FALSE;
						EDTXV2119.input.auto_open_signal := FALSE;
						EDTXV2126.input.auto_open_signal := FALSE;
						EDTXV2113.input.auto_open_signal := FALSE;
						EDTXV2107.input.auto_open_signal := FALSE;
						EDTR20.input.auto_run_signal := FALSE;
						IF EDTXV2107.input.close_feedback_state AND EDTXV2113.input.close_feedback_state AND EDTXV2119.input.close_feedback_state AND
							EDTXV2126.input.close_feedback_state AND (NOT EDTP34.input.run_feedback) AND (NOT EDTR20.input.run_feedback)THEN
							EDTP3S3C_STEP[4].done := TRUE;
							p3_step3_4c := 0;
						END_IF;
				END_CASE;
				TON_23();
			5:
			//现场关闭P34循环水手阀
			EDTXV2127.input.auto_open_signal := FALSE;
		END_CASE;
	END_IF;

	//人工确认步骤可用
	IF (EDTP3S3C.status.run_state) AND (NOT EDTP3S3C_STEP[EDTP3S3C.status.run_step].done AND ((EDTP3S3C.status.run_step = 2) OR (EDTP3S3C.status.run_step = 5))) THEN
		EDTP3S3C.status.confirm_enable := TRUE;
	ELSE
		EDTP3S3C.status.confirm_enable := FALSE;
	END_IF;
END_ACTION

(* ---- EDTP4S1A_ACTION.st ---- *)
ACTION P4S1A_ACT:
	//设定时间
	FOR i := 0 TO EDTP4S1_STEP_NUM DO
		IF EDTP4S1A_ST[i] < T#5s THEN
			EDTP4S1A_ST[i] := T#5s;
		END_IF;
		EDTP4S1A_STEP[i].set_time := EDTP4S1A_ST[i];
	END_FOR;

	//流程步骤
	ProcessHandleFC(EDTP4S1A,EDTP4S1A_STEP[0],EDTP4S1_STEP_NUM);

	//object 手自动切换
	IF (EDTP4S1A.status.mode <> 0) AND (NOT EDTP4S1A.auto_mode_edge) THEN
		EDTP4S1A.auto_mode_edge := TRUE;
		EDTP4S1A.manual_mode_edge := FALSE;

		EDTXV1011.control.auto_operate := TRUE;
		EDTXV1009.control.auto_operate := TRUE;
		EDTP16.control.auto_operate := TRUE;
		EDTLV1002.control.auto_operate := TRUE;
		STFP06.control.auto_operate := TRUE;
		STFLV0602.control.auto_operate := TRUE;
		STFLV0601.control.auto_operate := TRUE;
		EDTLV1003.control.auto_operate := TRUE;
		EDTFQV1001A.control.auto_operate := TRUE;
		EDTTV1002B.control.auto_operate := TRUE;
		EDTXV1010.control.auto_operate := TRUE;
		EDTXV1003.control.auto_operate := TRUE;
		EDTTV1001A.control.auto_operate := TRUE;
		EDTTV1001B.control.auto_operate := TRUE;
		EDTTV1002A.control.auto_operate := TRUE;
		EDTXV1006.control.auto_operate := TRUE;
		EDTR04A.control.auto_operate := TRUE;
		EDTLV1004A.control.auto_operate := TRUE;
	END_IF;

	IF (EDTP4S1A.status.mode = 0) AND (NOT EDTP4S1A.manual_mode_edge) THEN
		EDTP4S1A.manual_mode_edge := TRUE;
		EDTP4S1A.auto_mode_edge := FALSE;

		EDTXV1011.control.manual_operate := TRUE;
		EDTXV1009.control.manual_operate := TRUE;
		EDTP16.control.manual_operate := TRUE;
		EDTLV1002.control.manual_operate := TRUE;
		STFP06.control.manual_operate := TRUE;
		STFLV0602.control.manual_operate := TRUE;
		STFLV0601.control.manual_operate := TRUE;
		EDTLV1003.control.manual_operate := TRUE;
		EDTFQV1001A.control.manual_operate := TRUE;
		EDTTV1002B.control.manual_operate := TRUE;
		EDTXV1010.control.manual_operate := TRUE;
		EDTXV1003.control.manual_operate := TRUE;
		EDTTV1001A.control.manual_operate := TRUE;
		EDTTV1001B.control.manual_operate := TRUE;
		EDTTV1002A.control.manual_operate := TRUE;
		EDTXV1006.control.manual_operate := TRUE;
		EDTR04A.control.manual_operate := TRUE;
		EDTLV1004A.control.manual_operate := TRUE;
	END_IF;

	//错误信号停机
	EDTP4S1A.input.error_signal := (EDTXV1011.status.valve_status >= 2) OR
	(EDTXV1009.status.valve_status >= 2) OR (EDTP16.status.motor_status >= 2) OR
	(EDTLV1002.status.valve_status >= 2) OR (STFP06.status.motor_status >= 2) OR (STFLV0602.status.valve_status >= 2) OR
	(STFLV0601.status.valve_status >= 2) OR (EDTLV1003.status.valve_status >= 2) OR (EDTFQV1001A.status.valve_status >= 2) OR
	(EDTTV1002B.status.valve_status >= 2) OR (EDTXV1010.status.valve_status >= 2) OR
	(EDTXV1003.status.valve_status >= 2) OR (EDTTV1001A.status.valve_status >= 2) OR (EDTTV1001B.status.valve_status >= 2) OR
	(EDTTV1002A.status.valve_status >= 2) OR (EDTR04A.status.motor_status >= 2) OR (EDTXV1006.status.valve_status >= 2);

	//EDTLV1004A自动补水
	//	IF EDTTIT1001.status.value >= EDTP4S1A_PARA_Temp7 THEN
	//		EDTLV1004A.input.auto_open_signal := TRUE;
	//	ELSIF EDTTIT1001.status.value <= (EDTP4S1A_PARA_Temp7 - EDTP4S1A_PARA_Temp8) THEN
	//		EDTLV1004A.input.auto_open_signal := FALSE;
	//	END_IF;
	IF r04a_water THEN
		CASE r04a_water_step OF
			0:
				EDTLV1004A.control.auto_operate := TRUE;
				r04a_water_step := 1;
			1:
				EDTLV1004A.input.auto_open_signal := TRUE;
				r04a_temp := EDTTIT1001.status.value;
				r04a_water_step := 2;
			2:
				IF r04a_temp - EDTTIT1001.status.value >= EDTP4S1A_PARA_Temp8 THEN
					EDTLV1004A.input.auto_open_signal := FALSE;
					r04a_water_step := 0;
					r04a_water := FALSE;
				END_IF;
		END_CASE;
	END_IF;

	IF EDTP4S1A.status.run_state = 1 THEN
		CASE EDTP4S1A.status.run_step OF
			0:
				IF NOT EDTP4S1A_STEP[0].done THEN
					EDTXV1011.control.auto_operate := TRUE;
					EDTXV1009.control.auto_operate := TRUE;
					EDTP16.control.auto_operate := TRUE;
					EDTLV1002.control.auto_operate := TRUE;
					STFP06.control.auto_operate := TRUE;
					STFLV0602.control.auto_operate := TRUE;
					STFLV0601.control.auto_operate := TRUE;
					EDTLV1003.control.auto_operate := TRUE;
					EDTFQV1001A.control.auto_operate := TRUE;
					EDTTV1002B.control.auto_operate := TRUE;
					EDTXV1010.control.auto_operate := TRUE;
					EDTXV1003.control.auto_operate := TRUE;
					EDTTV1001A.control.auto_operate := TRUE;
					EDTTV1001B.control.auto_operate := TRUE;
					EDTTV1002A.control.auto_operate := TRUE;
					EDTXV1006.control.auto_operate := TRUE;
					EDTR04A.control.auto_operate := TRUE;
					EDTLV1004A.control.auto_operate := TRUE;
					EDTP4S1A_STEP[0].done := TRUE;
				END_IF;
			1:
				//手动进DMSO和纯水
			2:
				EDTTV1001A.input.auto_open_signal := TRUE;
				EDTTV1001B.input.auto_open_signal := TRUE;
				EDTXV1010.input.auto_open_signal := TRUE;
				EDTXV1003.input.auto_open_signal := TRUE;
				EDTR04A.input.auto_run_signal := TRUE;
				EDTTV1002B.input.auto_open_signal := TRUE;
				EDTXV1006.input.auto_open_signal := TRUE;
				IF EDTXV1010.input.open_feedback_state AND EDTXV1003.input.open_feedback_state AND EDTR04A.input.run_feedback
					AND EDTTV1002B.input.open_feedback_state AND EDTXV1006.input.open_feedback_state THEN
					EDTP4S1A_STEP[2].done := TRUE;
				END_IF;
			3:
				CASE p4_step1_3a OF
					0:
						IF NOT EDTP4S1A_STEP[3].done THEN
							p4_step1_3a := 1;
						END_IF;
					1:
						R04A_heat := TRUE;
						p4_step1_3a := 2;
					2:
						IF EDTTIT1001.status.value >= EDTP4S1A_PARA_Temp1 THEN
							EDTTV1002B.input.auto_open_signal := FALSE;
							IF EDTTV1002B.input.close_feedback_state THEN
								EDTTV1002A.input.auto_open_signal := TRUE;
								IF EDTTV1002A.input.open_feedback_state THEN
									p4_step1_3a := 3;
								END_IF;
							END_IF;
						END_IF;
					3:
						TON_63.PT := DINT_TO_TIME(EDTP4S1A_PARA_T4 * 3600 * 1000);
						IF EDTTIT1001.status.value >= EDTP4S1A_PARA_Temp2 THEN
							R04A_heat := FALSE;
							R04A_hold := TRUE;
							TON_63.IN := TRUE;
						END_IF;
						IF TON_63.Q THEN
							TON_63.IN := FALSE;
							p4_step1_3a := 4;
						END_IF;
					4:
						p4_step1_3a := 0;
						EDTP4S1A_STEP[3].done := TRUE;
				END_CASE;
				TON_63();
			4:
				//人工取样,确认反应结束
			5:
				R04A_hold := FALSE;
				EDTTV1001A.input.auto_open_signal := FALSE;
				EDTTV1001B.input.auto_open_signal := FALSE;
				IF EDTTV1001A.input.close_feedback_state AND EDTTV1001B.input.close_feedback_state THEN
					EDTP4S1A_STEP[5].done := TRUE;
				END_IF;
			6:
				IF EDTTIT1001.status.value <= EDTP4S1A_PARA_Temp5 THEN
					//					EDTXV1010.input.auto_open_signal := FALSE;
					//					EDTXV1003.input.auto_open_signal := FALSE;
					EDTTV1002A.input.auto_open_signal := FALSE;
				END_IF;
				IF (*EDTXV1010.input.close_feedback_state AND EDTXV1003.input.close_feedback_state AND *)(NOT EDTR04A.input.run_feedback)
					AND EDTTV1002A.input.close_feedback_state THEN
					EDTP4S1A_STEP[6].done := TRUE;
				END_IF;
			7:
				//转移
			8:
				EDTR04A.input.auto_run_signal := FALSE;
				IF NOT EDTR04A.input.run_feedback THEN
					EDTP4S1A_STEP[8].done := TRUE;
				END_IF;
		END_CASE;
	END_IF;

	Slope_0(value := EDTTIT1001.status.value, sample_time := EDTP4S1A_PARA_T5);

	IF R04A_heat THEN
		IF Slope_0.out <= EDTP4S1A_PARA_Slope1 THEN
			EDTTV1001A.input.auto_open_signal := TRUE;
			EDTTV1001B.input.auto_open_signal := TRUE;
		END_IF;
		IF Slope_0.out > EDTP4S1A_PARA_Slope1 AND Slope_0.out <= EDTP4S1A_PARA_Slope2 THEN
			EDTTV1001A.input.auto_open_signal := TRUE;
			EDTTV1001B.input.auto_open_signal := FALSE;
		END_IF;
		IF Slope_0.out > EDTP4S1A_PARA_Slope2 AND Slope_0.out <= EDTP4S1A_PARA_Slope3 THEN
			EDTTV1001A.input.auto_open_signal := FALSE;
			EDTTV1001B.input.auto_open_signal := TRUE;
		END_IF;
		IF Slope_0.out > EDTP4S1A_PARA_Slope3 THEN
			EDTTV1001A.input.auto_open_signal := FALSE;
			EDTTV1001B.input.auto_open_signal := FALSE;
		END_IF;
	END_IF;

	//155-158 大  158-162小阀 162都关
	IF R04A_hold THEN
		IF EDTTIT1001.status.value < EDTP4S1A_PARA_Temp2 THEN
			EDTTV1001A.input.auto_open_signal := TRUE;
			EDTTV1001B.input.auto_open_signal := TRUE;
		END_IF;
		IF EDTTIT1001.status.value < EDTP4S1A_PARA_Temp3 AND EDTTIT1001.status.value >= (EDTP4S1A_PARA_Temp2 + EDTP4S1A_PARA_Temp6) THEN
			EDTTV1001A.input.auto_open_signal := TRUE;
			EDTTV1001B.input.auto_open_signal := FALSE;
		END_IF;
		IF EDTTIT1001.status.value < EDTP4S1A_PARA_Temp4 AND EDTTIT1001.status.value >= (EDTP4S1A_PARA_Temp3 + EDTP4S1A_PARA_Temp6) THEN
			EDTTV1001A.input.auto_open_signal := FALSE;
			EDTTV1001B.input.auto_open_signal := TRUE;
		END_IF;
		IF EDTTIT1001.status.value >= (EDTP4S1A_PARA_Temp4 + EDTP4S1A_PARA_Temp6) THEN
			EDTTV1001A.input.auto_open_signal := FALSE;
			EDTTV1001B.input.auto_open_signal := FALSE;
		END_IF;
	END_IF;

	//======================================================================================================
	//DMSO进料
	//从罐区进料
	IF pot_to_r04_a THEN
		CASE pot_to_r04_a_step OF
			0:
				EDTFQV1001A.input.auto_open_signal := TRUE;
				EDTLV1003.input.auto_open_signal := TRUE;
				STFLV0601.input.auto_open_signal := FALSE;
				STFLV0602.input.auto_open_signal := FALSE;
				(*IF EDTFQV1001A.input.open_feedback_state AND*)IF EDTLV1003.input.open_feedback_state AND//note:反馈有问题，临时去掉EDTFQV1001A
					STFLV0601.input.close_feedback_state AND STFLV0602.input.close_feedback_state THEN
					pot_to_r04_a_step := 1;
				END_IF;
			1:
				LiquidTransfer_28(sp_time := DINT_TO_TIME(EDTP4S1A_PARA_T2 * 1000),
				sp_accumulation := EDTP4S1A_PARA_AC1,
				done := pot_to_r04_a_step_1_done,
				flowmeter := EDTFQIT1001);
				STFP06.input.auto_run_signal := LiquidTransfer_28.run;
				IF pot_to_r04_a_step_1_done AND (NOT STFP06.input.run_feedback) AND (NOT STFP06.input.auto_run_signal) THEN
					pot_to_r04_a_step_1_done := FALSE;
					pot_to_r04_a_step := 2;
				END_IF;
			2:
				IF EDTFQIT1001.flowrate <= flowrate_threshold THEN
					pot_to_r04_a_step := 3;
				END_IF;
			3:
				EDTFQV1001A.input.auto_open_signal := FALSE;
				EDTLV1003.input.auto_open_signal := FALSE;
				IF EDTFQV1001A.input.close_feedback_state AND EDTLV1003.input.close_feedback_state THEN
					pot_to_r04_a_step := 0;
					pot_to_r04_a := FALSE;
				END_IF;
		END_CASE;
	END_IF;

	//从V52进料
	IF v52_to_r04_a THEN
		CASE v52_to_r04_a_step OF
			0:
				EDTFQV1001A.input.auto_open_signal := TRUE;
				EDTLV1002.input.auto_open_signal := TRUE;
				(*IF EDTFQV1001A.input.open_feedback_state AND*)IF EDTLV1002.input.open_feedback_state THEN
					v52_to_r04_a_step := 1;
				END_IF;
			1:
				LiquidTransfer_29(sp_time := DINT_TO_TIME(EDTP4S1A_PARA_T3 * 1000),
				sp_accumulation := EDTP4S1A_PARA_AC2,
				done := v52_to_r04_a_step_1_done,
				flowmeter := EDTFQIT1001);
				EDTP16.input.auto_run_signal := LiquidTransfer_29.run;
				IF v52_to_r04_a_step_1_done AND (NOT EDTP16.input.run_feedback) AND (NOT EDTP16.input.auto_run_signal) THEN
					v52_to_r04_a_step_1_done := FALSE;
					v52_to_r04_a_step := 2;
				END_IF;
			2:
				IF EDTFQIT1001.flowrate <= flowrate_threshold THEN
					v52_to_r04_a_step := 3;
				END_IF;
			3:
				EDTFQV1001A.input.auto_open_signal := FALSE;
				EDTLV1002.input.auto_open_signal := FALSE;
				IF EDTFQV1001A.input.close_feedback_state AND EDTLV1002.input.close_feedback_state THEN
					v52_to_r04_a_step := 0;
					v52_to_r04_a := FALSE;
				END_IF;
		END_CASE;
	END_IF;

	//=======================================================================================================
	//人工确认步骤可用
	IF (EDTP4S1A.status.run_state) AND (NOT EDTP4S1A_STEP[EDTP4S1A.status.run_step].done AND ((EDTP4S1A.status.run_step = 1) OR (EDTP4S1A.status.run_step = 4) OR (EDTP4S1A.status.run_step = 7))) THEN
		EDTP4S1A.status.confirm_enable := TRUE;
	ELSE
		EDTP4S1A.status.confirm_enable := FALSE;
	END_IF;
END_ACTION

(* ---- EDTP4S1B_ACTION.st ---- *)
ACTION P4S1B_ACT:
	//设定时间
	FOR i := 0 TO EDTP4S1_STEP_NUM DO
		IF EDTP4S1B_ST[i] < T#5s THEN
			EDTP4S1B_ST[i] := T#5s;
		END_IF;
		EDTP4S1B_STEP[i].set_time := EDTP4S1B_ST[i];
	END_FOR;

	//流程步骤
	ProcessHandleFC(EDTP4S1B,EDTP4S1B_STEP[0],EDTP4S1_STEP_NUM);

	//object 手自动切换
	IF (EDTP4S1B.status.mode <> 0) AND (NOT EDTP4S1B.auto_mode_edge) THEN
		EDTP4S1B.auto_mode_edge := TRUE;
		EDTP4S1B.manual_mode_edge := FALSE;

		EDTXV1011.control.auto_operate := TRUE;
		EDTXV1009.control.auto_operate := TRUE;
		EDTP16.control.auto_operate := TRUE;
		EDTLV1002.control.auto_operate := TRUE;
		STFP06.control.auto_operate := TRUE;
		STFLV0602.control.auto_operate := TRUE;
		STFLV0601.control.auto_operate := TRUE;
		EDTLV1003.control.auto_operate := TRUE;
		EDTFQV1001B.control.auto_operate := TRUE;
		EDTTV1004B.control.auto_operate := TRUE;
		EDTXV1015.control.auto_operate := TRUE;
		EDTXV1013.control.auto_operate := TRUE;
		EDTTV1003A.control.auto_operate := TRUE;
		EDTTV1003B.control.auto_operate := TRUE;
		EDTTV1004A.control.auto_operate := TRUE;
		EDTXV1014.control.auto_operate := TRUE;
		EDTR04B.control.auto_operate := TRUE;
		EDTLV1004B.control.auto_operate := TRUE;
	END_IF;

	IF (EDTP4S1B.status.mode = 0) AND (NOT EDTP4S1B.manual_mode_edge) THEN
		EDTP4S1B.manual_mode_edge := TRUE;
		EDTP4S1B.auto_mode_edge := FALSE;

		EDTXV1011.control.manual_operate := TRUE;
		EDTXV1009.control.manual_operate := TRUE;
		EDTP16.control.manual_operate := TRUE;
		EDTLV1002.control.manual_operate := TRUE;
		STFP06.control.manual_operate := TRUE;
		STFLV0602.control.manual_operate := TRUE;
		STFLV0601.control.manual_operate := TRUE;
		EDTLV1003.control.manual_operate := TRUE;
		EDTFQV1001B.control.manual_operate := TRUE;
		EDTTV1004B.control.manual_operate := TRUE;
		EDTXV1015.control.manual_operate := TRUE;
		EDTXV1013.control.manual_operate := TRUE;
		EDTTV1003A.control.manual_operate := TRUE;
		EDTTV1003B.control.manual_operate := TRUE;
		EDTTV1004A.control.manual_operate := TRUE;
		EDTXV1014.control.manual_operate := TRUE;
		EDTR04B.control.manual_operate := TRUE;
		EDTLV1004B.control.manual_operate := TRUE;
	END_IF;

	//错误信号停机
	EDTP4S1B.input.error_signal := (EDTXV1011.status.valve_status >= 2) OR
	(EDTXV1009.status.valve_status >= 2) OR (EDTP16.status.motor_status >= 2) OR
	(EDTLV1002.status.valve_status >= 2) OR (STFP06.status.motor_status >= 2) OR (STFLV0602.status.valve_status >= 2) OR
	(STFLV0601.status.valve_status >= 2) OR (EDTLV1003.status.valve_status >= 2) OR (EDTFQV1001B.status.valve_status >= 2) OR
	(EDTTV1004B.status.valve_status >= 2) OR (EDTXV1015.status.valve_status >= 2) OR
	(EDTXV1013.status.valve_status >= 2) OR (EDTTV1003A.status.valve_status >= 2) OR (EDTTV1003B.status.valve_status >= 2) OR
	(EDTTV1004A.status.valve_status >= 2) OR (EDTR04B.status.motor_status >= 2) OR (EDTXV1014.status.valve_status >= 2);

	//EDTLV1004B自动补水
	//	IF EDTTIT1003.status.value >= EDTP4S1B_PARA_Temp7 THEN
	//		EDTLV1004B.input.auto_open_signal := TRUE;
	//	ELSIF EDTTIT1003.status.value <= (EDTP4S1B_PARA_Temp7 - EDTP4S1B_PARA_Temp8) THEN
	//		EDTLV1004B.input.auto_open_signal := FALSE;
	//	END_IF;
	IF r04b_water THEN
		CASE r04b_water_step OF
			0:
				EDTLV1004B.control.auto_operate := TRUE;
				r04b_water_step := 1;
			1:
				EDTLV1004B.input.auto_open_signal := TRUE;
				r04b_temp := EDTTIT1003.status.value;
				r04b_water_step := 2;
			2:
				IF r04b_temp - EDTTIT1003.status.value >= EDTP4S1B_PARA_Temp8 THEN
					EDTLV1004B.input.auto_open_signal := FALSE;
					r04b_water_step := 0;
					r04b_water := FALSE;
				END_IF;
		END_CASE;
	END_IF;

	IF EDTP4S1B.status.run_state = 1 THEN
		CASE EDTP4S1B.status.run_step OF
			0:
				IF NOT EDTP4S1B_STEP[0].done THEN
					EDTXV1011.control.auto_operate := TRUE;
					EDTXV1009.control.auto_operate := TRUE;
					EDTP16.control.auto_operate := TRUE;
					EDTLV1002.control.auto_operate := TRUE;
					STFP06.control.auto_operate := TRUE;
					STFLV0602.control.auto_operate := TRUE;
					STFLV0601.control.auto_operate := TRUE;
					EDTLV1003.control.auto_operate := TRUE;
					EDTFQV1001B.control.auto_operate := TRUE;
					EDTTV1004B.control.auto_operate := TRUE;
					EDTXV1015.control.auto_operate := TRUE;
					EDTXV1013.control.auto_operate := TRUE;
					EDTTV1003A.control.auto_operate := TRUE;
					EDTTV1003B.control.auto_operate := TRUE;
					EDTTV1004A.control.auto_operate := TRUE;
					EDTXV1014.control.auto_operate := TRUE;
					EDTR04B.control.auto_operate := TRUE;
					EDTLV1004B.control.auto_operate := TRUE;
					EDTP4S1B_STEP[0].done := TRUE;
				END_IF;
			1:
				//手动进DMSO和纯水
			2:
				EDTTV1003A.input.auto_open_signal := TRUE;
				EDTTV1003B.input.auto_open_signal := TRUE;
				EDTXV1015.input.auto_open_signal := TRUE;
				EDTXV1013.input.auto_open_signal := TRUE;
				EDTR04B.input.auto_run_signal := TRUE;
				EDTTV1004B.input.auto_open_signal := TRUE;
				EDTXV1014.input.auto_open_signal := TRUE;
				IF EDTXV1015.input.open_feedback_state AND EDTXV1013.input.open_feedback_state AND EDTR04B.input.run_feedback
					AND EDTTV1004B.input.open_feedback_state AND EDTXV1014.input.open_feedback_state THEN
					EDTP4S1B_STEP[2].done := TRUE;
				END_IF;
			3:
				CASE p4_step1_3b OF
					0:
						IF NOT EDTP4S1B_STEP[3].done THEN
							p4_step1_3b := 1;
						END_IF;
					1:
						R04B_heat := TRUE;
						p4_step1_3b := 2;
					2:
						IF EDTTIT1003.status.value >= EDTP4S1B_PARA_Temp1 THEN
							EDTTV1004B.input.auto_open_signal := FALSE;
							IF EDTTV1004B.input.close_feedback_state THEN
								EDTTV1004A.input.auto_open_signal := TRUE;
								IF EDTTV1004A.input.open_feedback_state THEN
									p4_step1_3b := 3;
								END_IF;
							END_IF;
						END_IF;
					3:
						TON_76.PT := DINT_TO_TIME(EDTP4S1B_PARA_T4 * 3600 * 1000);
						IF EDTTIT1003.status.value >= EDTP4S1B_PARA_Temp2 THEN
							R04B_heat := FALSE;
							R04B_hold := TRUE;
							TON_76.IN := TRUE;
						END_IF;
						IF TON_76.Q THEN
							TON_76.IN := FALSE;
							p4_step1_3b := 4;
						END_IF;
					4:
						p4_step1_3b := 0;
						EDTP4S1B_STEP[3].done := TRUE;
				END_CASE;
				TON_76();
			4:
				//人工取样,确认反应结束
			5:
				R04B_hold := FALSE;
				EDTTV1003A.input.auto_open_signal := FALSE;
				EDTTV1003B.input.auto_open_signal := FALSE;
				IF EDTTV1003A.input.close_feedback_state AND EDTTV1003B.input.close_feedback_state THEN
					EDTP4S1B_STEP[5].done := TRUE;
				END_IF;
			6:
				IF EDTTIT1003.status.value <= EDTP4S1B_PARA_Temp5 THEN
					//					EDTXV1015.input.auto_open_signal := FALSE;
					//					EDTXV1013.input.auto_open_signal := FALSE;
					EDTTV1004A.input.auto_open_signal := FALSE;
				END_IF;
				IF(* EDTXV1015.input.close_feedback_state AND EDTXV1013.input.close_feedback_state AND *)(NOT EDTR04B.input.run_feedback)
					AND EDTTV1004A.input.close_feedback_state THEN
					EDTP4S1B_STEP[6].done := TRUE;
				END_IF;
			7:
				//转移
			8:
				EDTR04B.input.auto_run_signal := FALSE;
				IF NOT EDTR04B.input.run_feedback THEN
					EDTP4S1B_STEP[8].done := TRUE;
				END_IF;

		END_CASE;
	END_IF;

	Slope_1(value := EDTTIT1003.status.value, sample_time := EDTP4S1B_PARA_T5);
	IF R04B_heat THEN
		IF Slope_1.out <= EDTP4S1B_PARA_Slope1 THEN
			EDTTV1003A.input.auto_open_signal := TRUE;
			EDTTV1003B.input.auto_open_signal := TRUE;
		END_IF;
		IF Slope_1.out > EDTP4S1B_PARA_Slope1 AND Slope_1.out <= EDTP4S1B_PARA_Slope2 THEN
			EDTTV1003A.input.auto_open_signal := TRUE;
			EDTTV1003B.input.auto_open_signal := FALSE;
		END_IF;
		IF Slope_1.out > EDTP4S1B_PARA_Slope2 AND Slope_1.out <= EDTP4S1B_PARA_Slope3 THEN
			EDTTV1003A.input.auto_open_signal := FALSE;
			EDTTV1003B.input.auto_open_signal := TRUE;
		END_IF;
		IF Slope_1.out > EDTP4S1B_PARA_Slope3 THEN
			EDTTV1003A.input.auto_open_signal := FALSE;
			EDTTV1003B.input.auto_open_signal := FALSE;
		END_IF;
	END_IF;

	//155-158 大  158-162小阀 162都关
	IF R04B_hold THEN
		IF EDTTIT1003.status.value < EDTP4S1B_PARA_Temp2 THEN
			EDTTV1003A.input.auto_open_signal := TRUE;
			EDTTV1003B.input.auto_open_signal := TRUE;
		END_IF;
		IF EDTTIT1003.status.value < EDTP4S1B_PARA_Temp3 AND EDTTIT1003.status.value >= (EDTP4S1B_PARA_Temp2 + EDTP4S1B_PARA_Temp6) THEN
			EDTTV1003A.input.auto_open_signal := TRUE;
			EDTTV1003B.input.auto_open_signal := FALSE;
		END_IF;
		IF EDTTIT1003.status.value < EDTP4S1B_PARA_Temp4 AND EDTTIT1003.status.value >= (EDTP4S1B_PARA_Temp3 + EDTP4S1B_PARA_Temp6) THEN
			EDTTV1003A.input.auto_open_signal := FALSE;
			EDTTV1003B.input.auto_open_signal := TRUE;
		END_IF;
		IF EDTTIT1003.status.value >= (EDTP4S1B_PARA_Temp4 + EDTP4S1B_PARA_Temp6) THEN
			EDTTV1003A.input.auto_open_signal := FALSE;
			EDTTV1003B.input.auto_open_signal := FALSE;
		END_IF;
	END_IF;

	//======================================================================================================
	//DMSO进料
	//从罐区进料
	IF pot_to_r04_b THEN
		CASE pot_to_r04_b_step OF
			0:
				EDTFQV1001B.input.auto_open_signal := TRUE;
				EDTLV1003.input.auto_open_signal := TRUE;
				STFLV0601.input.auto_open_signal := FALSE;
				STFLV0602.input.auto_open_signal := FALSE;
				IF EDTFQV1001B.input.open_feedback_state AND EDTLV1003.input.open_feedback_state AND
					STFLV0601.input.close_feedback_state AND STFLV0602.input.close_feedback_state THEN
					pot_to_r04_b_step := 1;
				END_IF;
			1:
				LiquidTransfer_11(sp_time := DINT_TO_TIME(EDTP4S1B_PARA_T2 * 1000),
				sp_accumulation := EDTP4S1B_PARA_AC1,
				done := pot_to_r04_b_step_1_done,
				flowmeter := EDTFQIT1001);
				STFP06.input.auto_run_signal := LiquidTransfer_11.run;
				IF pot_to_r04_b_step_1_done AND (NOT STFP06.input.run_feedback) AND (NOT STFP06.input.auto_run_signal) THEN
					pot_to_r04_b_step_1_done := FALSE;
					pot_to_r04_b_step := 2;
				END_IF;
			2:
				IF EDTFQIT1001.flowrate <= flowrate_threshold THEN
					pot_to_r04_b_step := 3;
				END_IF;
			3:
				EDTFQV1001B.input.auto_open_signal := FALSE;
				EDTLV1003.input.auto_open_signal := FALSE;
				IF EDTFQV1001B.input.close_feedback_state AND EDTLV1003.input.close_feedback_state THEN
					pot_to_r04_b_step := 0;
					pot_to_r04_b := FALSE;
				END_IF;
		END_CASE;
	END_IF;

	//从V52进料
	IF v52_to_r04_b THEN
		CASE v52_to_r04_b_step OF
			0:
				EDTFQV1001B.input.auto_open_signal := TRUE;
				EDTLV1002.input.auto_open_signal := TRUE;
				IF EDTFQV1001B.input.open_feedback_state AND EDTLV1002.input.open_feedback_state THEN
					v52_to_r04_b_step := 1;
				END_IF;
			1:
				LiquidTransfer_14(sp_time := DINT_TO_TIME(EDTP4S1B_PARA_T3 * 1000),
				sp_accumulation := EDTP4S1B_PARA_AC2,
				done := v52_to_r04_b_step_1_done,
				flowmeter := EDTFQIT1001);
				EDTP16.input.auto_run_signal := LiquidTransfer_14.run;
				IF v52_to_r04_b_step_1_done AND (NOT EDTP16.input.run_feedback) AND (NOT EDTP16.input.auto_run_signal) THEN
					v52_to_r04_b_step_1_done := FALSE;
					v52_to_r04_b_step := 2;
				END_IF;
			2:
				IF EDTFQIT1001.flowrate <= flowrate_threshold THEN
					v52_to_r04_b_step := 3;
				END_IF;
			3:
				EDTFQV1001B.input.auto_open_signal := FALSE;
				EDTLV1002.input.auto_open_signal := FALSE;
				IF EDTFQV1001B.input.close_feedback_state AND EDTLV1002.input.close_feedback_state THEN
					v52_to_r04_b_step := 0;
					v52_to_r04_b := FALSE;
				END_IF;
		END_CASE;
	END_IF;

	//=======================================================================================================
	//人工确认步骤可用
	IF (EDTP4S1B.status.run_state) AND (NOT EDTP4S1B_STEP[EDTP4S1B.status.run_step].done AND ((EDTP4S1B.status.run_step = 1) OR (EDTP4S1B.status.run_step = 4) OR (EDTP4S1B.status.run_step = 7))) THEN
		EDTP4S1B.status.confirm_enable := TRUE;
	ELSE
		EDTP4S1B.status.confirm_enable := FALSE;
	END_IF;
END_ACTION
